(* CoDeSys 2.3.9.47 project: 3floor_2016_06_22_beta.prx *)
(* Libraries: TcEIB.lbx 16.5.14 14:12:22, TcSystemBX.lbx 11.6.12 13:56:16, TcBaseBX.lbx 10.5.06 08:50:20, standard.lbx 5.12.03 08:02:30 *)

(* Task configuration *)
TASK Standard (PRIORITY := 0, INTERVAL := T#20ms);
	MAIN
END_TASK

(* Global variable list: M_Var_1 *)
VAR_GLOBAL

	komora_l_adr: 				EIB_GROUP_ADDR:= (MAIN:=1, SUB_MAIN:=1, NUMBER:=10);
	su1_l_adr: 					EIB_GROUP_ADDR:= (MAIN:=1, SUB_MAIN:=1, NUMBER:=11);
	topochna_l_adr:	 			EIB_GROUP_ADDR:= (MAIN:=1, SUB_MAIN:=1, NUMBER:=12);
	su2_bra_adr:	 			EIB_GROUP_ADDR:= (MAIN:=1, SUB_MAIN:=1, NUMBER:=13);
	su2_l_adr:	 				EIB_GROUP_ADDR:= (MAIN:=1, SUB_MAIN:=1, NUMBER:=14);
	su1_rakovyna_adr:	 		EIB_GROUP_ADDR:= (MAIN:=1, SUB_MAIN:=1, NUMBER:=15);
	su2_dush_adr:	 			EIB_GROUP_ADDR:= (MAIN:=1, SUB_MAIN:=1, NUMBER:=16);
	dush_adr:	 				EIB_GROUP_ADDR:= (MAIN:=1, SUB_MAIN:=1, NUMBER:=17);
	kuhnya1_adr:	 			EIB_GROUP_ADDR:= (MAIN:=1, SUB_MAIN:=1, NUMBER:=18);
	vitalnya_smugy1_adr: 		EIB_GROUP_ADDR:= (MAIN:=1, SUB_MAIN:=1, NUMBER:=19);
	vitalnya_l_adr: 				EIB_GROUP_ADDR:= (MAIN:=1, SUB_MAIN:=1, NUMBER:=20);
	vitalnya_prokladka_adr: 		EIB_GROUP_ADDR:= (MAIN:=1, SUB_MAIN:=1, NUMBER:=21);
	terassa_stina_adr: 			EIB_GROUP_ADDR:= (MAIN:=1, SUB_MAIN:=1, NUMBER:=22);
	pidval_shody_adr: 			EIB_GROUP_ADDR:= (MAIN:=1, SUB_MAIN:=1, NUMBER:=23);
	skhody2pov_adr: 			EIB_GROUP_ADDR:= (MAIN:=1, SUB_MAIN:=1, NUMBER:=24);
	tambur_l_adr:				EIB_GROUP_ADDR:= (MAIN:=1, SUB_MAIN:=1, NUMBER:=25);
	vent_su1_adr: 				EIB_GROUP_ADDR:= (MAIN:=1, SUB_MAIN:=1, NUMBER:=26);
	vent_kuh_low_adr: 			EIB_GROUP_ADDR:= (MAIN:=1, SUB_MAIN:=1, NUMBER:=27);
	vent_dush_adr: 				EIB_GROUP_ADDR:= (MAIN:=1, SUB_MAIN:=1, NUMBER:=28);
	vent_komora_adr: 			EIB_GROUP_ADDR:= (MAIN:=1, SUB_MAIN:=1, NUMBER:=29);
	vent_kuh_high_adr: 			EIB_GROUP_ADDR:= (MAIN:=1, SUB_MAIN:=1, NUMBER:=30);


	komora_l_status_adr: 				EIB_GROUP_ADDR:= (MAIN:=1, SUB_MAIN:=1, NUMBER:=110);
	su1_l_status_adr: 					EIB_GROUP_ADDR:= (MAIN:=1, SUB_MAIN:=1, NUMBER:=111);
	topochna_l_status_adr:	 			EIB_GROUP_ADDR:= (MAIN:=1, SUB_MAIN:=1, NUMBER:=112);
	su2_bra_status_adr:	 				EIB_GROUP_ADDR:= (MAIN:=1, SUB_MAIN:=1, NUMBER:=113);
	su2_l_status_adr:	 				EIB_GROUP_ADDR:= (MAIN:=1, SUB_MAIN:=1, NUMBER:=114);
	su1_rakovyna_status_adr:	 		EIB_GROUP_ADDR:= (MAIN:=1, SUB_MAIN:=1, NUMBER:=115);
	su2_dush_status_adr:	 			EIB_GROUP_ADDR:= (MAIN:=1, SUB_MAIN:=1, NUMBER:=116);
	dush_status_adr:	 				EIB_GROUP_ADDR:= (MAIN:=1, SUB_MAIN:=1, NUMBER:=117);
	kuhnya1_status_adr:	 				EIB_GROUP_ADDR:= (MAIN:=1, SUB_MAIN:=1, NUMBER:=118);
	vitalnya_smugy1_status_adr: 			EIB_GROUP_ADDR:= (MAIN:=1, SUB_MAIN:=1, NUMBER:=119);
	vitalnya_l_status_adr: 				EIB_GROUP_ADDR:= (MAIN:=1, SUB_MAIN:=1, NUMBER:=120);
	vitalnya_prokladka_status_adr: 		EIB_GROUP_ADDR:= (MAIN:=1, SUB_MAIN:=1, NUMBER:=121);
	terassa_stina_status_adr: 			EIB_GROUP_ADDR:= (MAIN:=1, SUB_MAIN:=1, NUMBER:=122);
	pidval_shody_status_adr: 			EIB_GROUP_ADDR:= (MAIN:=1, SUB_MAIN:=1, NUMBER:=123);
	skhody2pov_status_adr: 				EIB_GROUP_ADDR:= (MAIN:=1, SUB_MAIN:=1, NUMBER:=124);
	tambur_l_status_adr:					EIB_GROUP_ADDR:= (MAIN:=1, SUB_MAIN:=1, NUMBER:=125);
	vent_su1_status_adr: 				EIB_GROUP_ADDR:= (MAIN:=1, SUB_MAIN:=1, NUMBER:=126);
	vent_kuh_low_status_adr: 			EIB_GROUP_ADDR:= (MAIN:=1, SUB_MAIN:=1, NUMBER:=127);
	vent_dush_status_adr: 				EIB_GROUP_ADDR:= (MAIN:=1, SUB_MAIN:=1, NUMBER:=128);
	vent_komora_status_adr: 			EIB_GROUP_ADDR:= (MAIN:=1, SUB_MAIN:=1, NUMBER:=129);
	vent_kuh_high_status_adr: 			EIB_GROUP_ADDR:= (MAIN:=1, SUB_MAIN:=1, NUMBER:=130);



	fb_komora_l_send_status_ex: 			EIB_BIT_SEND_EX;
	fb_su1_l_send_status_ex: 				EIB_BIT_SEND_EX;
	fb_topochna_l_send_status_ex: 			EIB_BIT_SEND_EX;
	fb_su2_bra_send_status_ex: 				EIB_BIT_SEND_EX;
	fb_topochna2_l_send_status_ex: 		EIB_BIT_SEND_EX;
	fb_su2_l_send_status_ex: 				EIB_BIT_SEND_EX;
	fb_su1_rakovyna_send_status_ex: 		EIB_BIT_SEND_EX;
	fb_su2_dush_send_status_ex: 			EIB_BIT_SEND_EX;
	fb_dush_send_status_ex: 				EIB_BIT_SEND_EX;
	fb_vitalnya_smugy2_send_status_ex: 		EIB_BIT_SEND_EX;
	fb_su2_polytsi_send_status_ex: 			EIB_BIT_SEND_EX;
	fb_kuhnya1_send_status_ex: 			EIB_BIT_SEND_EX;
	fb_kuhnya2_send_status_ex: 			EIB_BIT_SEND_EX;
	fb_vitalnya_smugy1_send_status_ex: 		EIB_BIT_SEND_EX;
	fb_vitalnya_l_send_status_ex: 			EIB_BIT_SEND_EX;
	fb_vitalnya_prokladka_send_status_ex: 	EIB_BIT_SEND_EX;
	fb_terassa_stina_send_status_ex: 		EIB_BIT_SEND_EX;
	fb_pidval_shody_send_status_ex: 		EIB_BIT_SEND_EX;
	fb_skhody2pov_send_status_ex: 			EIB_BIT_SEND_EX;
	fb_tambur_l_send_status_ex: 			EIB_BIT_SEND_EX;
	fb_vent_su1_send_status_ex: 			EIB_BIT_SEND_EX;
	fb_vent_kuh_low_send_status_ex: 		EIB_BIT_SEND_EX;
	fb_vent_dush_send_status_ex: 			EIB_BIT_SEND_EX;
	fb_vent_komora_send_status_ex: 		EIB_BIT_SEND_EX;
	fb_vent_kuh_high_send_status_ex: 		EIB_BIT_SEND_EX;

	fb_komora_l_read: 			EIB_BIT_REC;
	fb_su1_l_read: 				EIB_BIT_REC;
	fb_topochna_l_read: 		EIB_BIT_REC;
	fb_su2_bra_read: 			EIB_BIT_REC;
	fb_topochna2_l_read: 		EIB_BIT_REC;
	fb_su2_l_read: 				EIB_BIT_REC;
	fb_su1_rakovyna_read: 		EIB_BIT_REC;
	fb_su2_dush_read: 			EIB_BIT_REC;
	fb_dush_read: 				EIB_BIT_REC;
	fb_vitalnya_smugy2_read: 	EIB_BIT_REC;
	fb_su2_polytsi_read: 		EIB_BIT_REC;
	fb_kuhnya1_read: 			EIB_BIT_REC;
	fb_kuhnya2_read: 			EIB_BIT_REC;
	fb_vitalnya_smugy1_read: 	EIB_BIT_REC;
	fb_vitalnya_l_read: 			EIB_BIT_REC;
	fb_vitalnya_prokladka_read: 	EIB_BIT_REC;
	fb_terassa_stina_read: 		EIB_BIT_REC;
	fb_pidval_shody_read: 		EIB_BIT_REC;
	fb_skhody2pov_read: 		EIB_BIT_REC;
	fb_tambur_l_read: 			EIB_BIT_REC;
	fb_vent_su1_read: 			EIB_BIT_REC;
	fb_vent_kuh_low_read: 		EIB_BIT_REC;
	fb_vent_dush_read: 			EIB_BIT_REC;
	fb_vent_komora_read: 		EIB_BIT_REC;
	fb_vent_kuh_high_read: 		EIB_BIT_REC;

	moove_garderob				AT%MX100.0:BOOL;
	moove_tambur					AT%MX100.1:BOOL;
	moove_dytjacha					AT%MX100.2:BOOL;
	moove_spalnya					AT%MX100.3:BOOL;
	moove_korydor					AT%MX100.4:BOOL;
	moove_skhody					AT%MX100.5:BOOL;

	komora_l 						AT%MX100.0:BOOL;
	su1_l 							AT%MX100.1:BOOL;
	topochna_l 						AT%MX100.2:BOOL;
	su2_bra	 						AT%MX100.3:BOOL;
	su2_l 							AT%MX100.4:BOOL;
	su1_rakovyna 					AT%MX100.5:BOOL;
	su2_dush 						AT%MX100.6:BOOL;
	dush 							AT%MX100.7:BOOL;

	kuhnya1	 					AT%MX101.0:BOOL;
	vitalnya_smugy1 				AT%MX101.1:BOOL;
	vitalnya_l 						AT%MX101.2:BOOL;
	vitalnya_prokladka 				AT%MX101.3:BOOL;
	terassa_stina	 				AT%MX101.4:BOOL;
	pidval_shody	 				AT%MX101.5:BOOL;
	skhody2pov 					AT%MX101.6:BOOL;
	tambur_l 						AT%MX101.7:BOOL;

	vent_su1 						AT%MX102.0:BOOL;
	vent_kuh_low 					AT%MX102.1:BOOL;
	vent_dush 						AT%MX102.2:BOOL;
	vent_komora 					AT%MX102.3:BOOL;
	vent_kuh_high 					AT%MX102.4:BOOL;

END_VAR

(* Global variable list: M_Var_2 *)
VAR_GLOBAL
	balkon_peryla_adr: EIB_GROUP_ADDR:=(MAIN:=1, SUB_MAIN:=4, NUMBER:=9);
	kino_l_adr: EIB_GROUP_ADDR:= (MAIN:=1, SUB_MAIN:=4, NUMBER:=10);
	balkon_bra_adr:	 EIB_GROUP_ADDR:= (MAIN:=1, SUB_MAIN:=4, NUMBER:=11);
	kabinet_balkon_l_adr:	 EIB_GROUP_ADDR:= (MAIN:=1, SUB_MAIN:=4, NUMBER:=12);
	balkon_adr:	 EIB_GROUP_ADDR:= (MAIN:=1, SUB_MAIN:=4, NUMBER:=13);
	korydor1_adr:	 EIB_GROUP_ADDR:= (MAIN:=1, SUB_MAIN:=4, NUMBER:=14);
	kino_bra_adr:	 EIB_GROUP_ADDR:= (MAIN:=1, SUB_MAIN:=4, NUMBER:=15);
	korydor2_adr:	 EIB_GROUP_ADDR:= (MAIN:=1, SUB_MAIN:=4, NUMBER:=16);
	studio_pidsvitka_adr:	 EIB_GROUP_ADDR:= (MAIN:=1, SUB_MAIN:=4, NUMBER:=17);
	skhody2_3_adr:	 EIB_GROUP_ADDR:= (MAIN:=1, SUB_MAIN:=4, NUMBER:=18);
	studio_l_adr:	 EIB_GROUP_ADDR:= (MAIN:=1, SUB_MAIN:=4, NUMBER:=19);
	kabinet_pidsvitka_kolo_adr:	 EIB_GROUP_ADDR:= (MAIN:=1, SUB_MAIN:=4, NUMBER:=20);
	kabinet_svitlo_adr:	 EIB_GROUP_ADDR:= (MAIN:=1, SUB_MAIN:=4, NUMBER:=21);
	stend_adr:	 EIB_GROUP_ADDR:= (MAIN:=1, SUB_MAIN:=4, NUMBER:=22);
	kabinet_kobra_adr:	 EIB_GROUP_ADDR:= (MAIN:=1, SUB_MAIN:=4, NUMBER:=23);
	skhody_peryla_adr:	 EIB_GROUP_ADDR:= (MAIN:=1, SUB_MAIN:=4, NUMBER:=24);
	tambur2_adr:	 EIB_GROUP_ADDR:= (MAIN:=1, SUB_MAIN:=4, NUMBER:=25);

	fb_balkon_peryla_send: EIB_BIT_SEND_MANUAL;
	fb_kino_l_send:  EIB_BIT_SEND_manual;
	fb_balkon_bra_send: EIB_BIT_SEND_manual;
	fb_kabinet_balkon_l_send:  EIB_BIT_SEND_manual;
	fb_balkon_send:	EIB_BIT_SEND_manual;
	fb_korydor1_send:	 EIB_BIT_SEND_manual;
	fb_kino_bra_send:	EIB_BIT_SEND_manual;
	fb_korydor2_send:	EIB_BIT_SEND_manual;
	fb_studio_pidsvitka_send: EIB_BIT_SEND_MANUAL;
	fb_skhody2_3_send:	  EIB_BIT_SEND_MANUAL;
	fb_studio_l_send:	 EIB_BIT_SEND_manual;
	fb_kabinet_pidsvitka_kolo_send:	EIB_BIT_SEND_MANUAL;
	fb_kabinet_svitlo_send:	EIB_BIT_SEND_manual;
	fb_stend_send:  EIB_BIT_SEND_manual;
	fb_kabinet_kobra_send:  EIB_BIT_SEND_manual;
	fb_skhody_peryla_send:  EIB_BIT_SEND_MANUAL;
	fb_tambur2_send: EIB_BIT_SEND_MANUAL;
	fb_balkon_peryla_read: EIB_BIT_REC;
	fb_kino_l_read:  EIB_BIT_rec;
	fb_balkon_bra_read: EIB_BIT_rec;
	fb_kabinet_balkon_l_read:  EIB_BIT_rec;
	fb_balkon_read:	EIB_BIT_rec;
	fb_korydor1_read:	 EIB_BIT_rec;
	fb_kino_bra_read:	EIB_BIT_rec;
	fb_korydor2_read:	EIB_BIT_rec;
	fb_studio_pidsvitka_read: EIB_BIT_rec;
	fb_skhody2_3_read:	  EIB_BIT_REC;
	fb_studio_l_read:	 EIB_BIT_rec;
	fb_kabinet_pidsvitka_kolo_read:	EIB_BIT_REC;
	fb_kabinet_svitlo_read:	EIB_BIT_REC;
	fb_stend_read:  EIB_BIT_rec;
	fb_kabinet_kobra_read:  EIB_BIT_rec;
	fb_skhody_peryla_read:  EIB_BIT_REC;
	fb_tambur2_read: EIB_BIT_REC;


	eib_shtory_kino, eib_tul_kino: EIB_BIT_REC; (*ловлять в мережі смартбаса телеграмки для штор і тюлей*)
	eib_shtory_kabinet, eib_tul_kabinet: EIB_BIT_REC;

	fb_eib_shtory_kino_move:EIB_BIT_REC;
	fb_eib_shtory_kino_position:EIB_8BIT_SIGN_REC;
	fb_eib_shtory_kino_actualPosition:EIB_8BIT_SIGN_SEND;

	fb_eib_tul_kino_move:EIB_BIT_REC;
	fb_eib_tul_kino_position:EIB_8BIT_SIGN_REC;
	fb_eib_tul_kino_actualPosition:EIB_8BIT_SIGN_SEND;

	fb_eib_shtory_kabinet_move:EIB_BIT_REC;
	fb_eib_shtory_kabinet_position:EIB_8BIT_SIGN_REC;
	fb_eib_shtory_kabinet_actualPosition:EIB_8BIT_SIGN_SEND;

	fb_eib_tul_kabinet_move:EIB_BIT_REC;
	fb_eib_tul_kabinet_position:EIB_8BIT_SIGN_REC;
	fb_eib_tul_kabinet_actualPosition:EIB_8BIT_SIGN_SEND;



	balkon_peryla					AT%MX200.0:BOOL;
	kino_l							AT%MX200.1:BOOL;
	balkon_bra						AT%MX200.2:BOOL;
	kabinet_balkon_l					AT%MX200.3:BOOL;
	balkon							AT%MX200.4:BOOL;
	korydor1							AT%MX200.5:BOOL;
	kino_bra							AT%MX200.6:BOOL;
	korydor2							AT%MX200.7:BOOL;
	studio_pidsvitka					AT%MX201.0:BOOL;
	skhody2_3						AT%MX201.1:BOOL;
	studio_l							AT%MX201.2:BOOL;
	kabinet_pidsvitka_kolo				AT%MX201.3:BOOL;
	kabinet_svitlo						AT%MX201.4:BOOL;
	kabinet_kobra					AT%MX201.5:BOOL;
	tambur2							AT%MX201.6:BOOL;
	stend							AT%MX201.7:BOOL;
	skhody_peryla					AT%MX202.0:BOOL;

	kino_shtory_status					AT%MX202.1:BOOL;
	kino_tul_status					AT%MX202.2:BOOL;
	kabinet_shtory_status				AT%MX202.3:BOOL;
	kabinet_tul_status					AT%MX202.4:BOOL;

	collector_kabinet1					AT%MX203.0:BOOL;
	collector_kabinet2					AT%MX203.1:BOOL;
	collector_studio1					AT%MX203.2:BOOL;
	collector_studio2					AT%MX203.3:BOOL;

	fancoil_kabinet_low				AT%MX203.4:BOOL;
	fancoil_kabinet_med				AT%MX203.5:BOOL;
	fancoil_kabinet_high				AT%MX203.6:BOOL;

	fancoil_kino_low					AT%MX203.7:BOOL;
	fancoil_kino_med					AT%MX204.0:BOOL;
	fancoil_kino_high					AT%MX204.1:BOOL;


	kino_shtory_ActualPosition		AT%MB205:USINT;
	kino_tul_ActualPosition			AT%MB206:USINT;
	kabinet_shtory_ActualPosition	AT%MB207:USINT;
	kabinet_tul_ActualPosition		AT%MB208:USINT;
END_VAR

(* Global variable list: M_Var_4 *)
VAR_GLOBAL

	derevo_vidpochynok1_adr:	 	EIB_GROUP_ADDR:= (MAIN:=1, SUB_MAIN:=7, NUMBER:=22);
	derevo_vidpochynok2_adr:	 	EIB_GROUP_ADDR:= (MAIN:=1, SUB_MAIN:=7, NUMBER:=1);
	derevo_veranda_adr:	 		EIB_GROUP_ADDR:= (MAIN:=1, SUB_MAIN:=7, NUMBER:=2);
	derevo_veranda_zovn_adr:	 	EIB_GROUP_ADDR:= (MAIN:=1, SUB_MAIN:=7, NUMBER:=3);
	derevo_vhid_zovn_adr:	 		EIB_GROUP_ADDR:= (MAIN:=1, SUB_MAIN:=7, NUMBER:=4);
	derevo_sauna_adr:	 			EIB_GROUP_ADDR:= (MAIN:=1, SUB_MAIN:=7, NUMBER:=5);
	derevo_vhid_adr:				EIB_GROUP_ADDR:= (MAIN:=1, SUB_MAIN:=7, NUMBER:=6);
	derevo_kotel_adr:		 		EIB_GROUP_ADDR:= (MAIN:=1, SUB_MAIN:=7, NUMBER:=7);
	derevo_korydor_adr:		 		EIB_GROUP_ADDR:= (MAIN:=1, SUB_MAIN:=7, NUMBER:=8);
	derevo_sinna_adr:		 		EIB_GROUP_ADDR:= (MAIN:=1, SUB_MAIN:=7, NUMBER:=9);
	derevo_hamam_adr:		 		EIB_GROUP_ADDR:= (MAIN:=1, SUB_MAIN:=7, NUMBER:=10);
	derevo_kuhnya_adr:	 			EIB_GROUP_ADDR:= (MAIN:=1, SUB_MAIN:=7, NUMBER:=11);
	derevo_bassein1_adr:			EIB_GROUP_ADDR:= (MAIN:=1, SUB_MAIN:=7, NUMBER:=12);
	derevo_bassein_lampa_adr:		EIB_GROUP_ADDR:= (MAIN:=1, SUB_MAIN:=7, NUMBER:=13);
	derevo_spalnya2_adr:			EIB_GROUP_ADDR:= (MAIN:=1, SUB_MAIN:=7, NUMBER:=14);
	derevo_terassa_adr:				EIB_GROUP_ADDR:= (MAIN:=1, SUB_MAIN:=7, NUMBER:=15);
	derevo_dush_adr:	 			EIB_GROUP_ADDR:= (MAIN:=1, SUB_MAIN:=7, NUMBER:=16);
	derevo_wc_adr:					EIB_GROUP_ADDR:= (MAIN:=1, SUB_MAIN:=7, NUMBER:=17);
	derevo_spalnya_verh_adr:		EIB_GROUP_ADDR:= (MAIN:=1, SUB_MAIN:=7, NUMBER:=18);
	derevo_spalnya1_adr:			EIB_GROUP_ADDR:= (MAIN:=1, SUB_MAIN:=7, NUMBER:=19);
	derevo_spalnya_su_adr:			EIB_GROUP_ADDR:= (MAIN:=1, SUB_MAIN:=7, NUMBER:=20);
	derevo_garderob_adr:			EIB_GROUP_ADDR:= (MAIN:=1, SUB_MAIN:=7, NUMBER:=21);
	derevo_dush2_adr:				EIB_GROUP_ADDR:= (MAIN:=1, SUB_MAIN:=7, NUMBER:=23);

	derevo_vidpochynok1_status_adr:	 	EIB_GROUP_ADDR:= (MAIN:=1, SUB_MAIN:=7, NUMBER:=122);
	derevo_vidpochynok2_status_adr:	 	EIB_GROUP_ADDR:= (MAIN:=1, SUB_MAIN:=7, NUMBER:=101);
	derevo_veranda_status_adr:	 			EIB_GROUP_ADDR:= (MAIN:=1, SUB_MAIN:=7, NUMBER:=102);
	derevo_veranda_zovn_status_adr:	 	EIB_GROUP_ADDR:= (MAIN:=1, SUB_MAIN:=7, NUMBER:=103);
	derevo_vhid_zovn_status_adr:	 		EIB_GROUP_ADDR:= (MAIN:=1, SUB_MAIN:=7, NUMBER:=104);
	derevo_sauna_status_adr:	 			EIB_GROUP_ADDR:= (MAIN:=1, SUB_MAIN:=7, NUMBER:=105);
	derevo_vhid_status_adr:					EIB_GROUP_ADDR:= (MAIN:=1, SUB_MAIN:=7, NUMBER:=106);
	derevo_kotel_status_adr:		 		EIB_GROUP_ADDR:= (MAIN:=1, SUB_MAIN:=7, NUMBER:=107);
	derevo_korydor_status_adr:		 		EIB_GROUP_ADDR:= (MAIN:=1, SUB_MAIN:=7, NUMBER:=108);
	derevo_sinna_status_adr:		 		EIB_GROUP_ADDR:= (MAIN:=1, SUB_MAIN:=7, NUMBER:=109);
	derevo_hamam_status_adr:		 		EIB_GROUP_ADDR:= (MAIN:=1, SUB_MAIN:=7, NUMBER:=110);
	derevo_kuhnya_status_adr:	 			EIB_GROUP_ADDR:= (MAIN:=1, SUB_MAIN:=7, NUMBER:=111);
	derevo_bassein1_status_adr:				EIB_GROUP_ADDR:= (MAIN:=1, SUB_MAIN:=7, NUMBER:=112);
	derevo_bassein_lampa_status_adr:		EIB_GROUP_ADDR:= (MAIN:=1, SUB_MAIN:=7, NUMBER:=113);
	derevo_spalnya2_status_adr:				EIB_GROUP_ADDR:= (MAIN:=1, SUB_MAIN:=7, NUMBER:=114);
	derevo_terassa_status_adr:				EIB_GROUP_ADDR:= (MAIN:=1, SUB_MAIN:=7, NUMBER:=115);
	derevo_dush_status_adr:	 			EIB_GROUP_ADDR:= (MAIN:=1, SUB_MAIN:=7, NUMBER:=116);
	derevo_wc_status_adr:					EIB_GROUP_ADDR:= (MAIN:=1, SUB_MAIN:=7, NUMBER:=117);
	derevo_spalnya_verh_status_adr:		EIB_GROUP_ADDR:= (MAIN:=1, SUB_MAIN:=7, NUMBER:=118);
	derevo_spalnya1_status_adr:				EIB_GROUP_ADDR:= (MAIN:=1, SUB_MAIN:=7, NUMBER:=119);
	derevo_spalnya_su_status_adr:			EIB_GROUP_ADDR:= (MAIN:=1, SUB_MAIN:=7, NUMBER:=120);
	derevo_garderob_status_adr:				EIB_GROUP_ADDR:= (MAIN:=1, SUB_MAIN:=7, NUMBER:=121);
	derevo_dush2_status_adr:				EIB_GROUP_ADDR:= (MAIN:=1, SUB_MAIN:=7, NUMBER:=123);

	fb_derevo_vidpochynok1_send_status_ex: 		EIB_BIT_SEND_EX;
	fb_derevo_vidpochynok2_send_status_ex: 		EIB_BIT_SEND_EX;
	fb_derevo_veranda_send_status_ex: 				EIB_BIT_SEND_EX;
	fb_derevo_veranda_zovn_send_status_ex: 		EIB_BIT_SEND_EX;
	fb_derevo_vhid_zovn_send_status_ex: 			EIB_BIT_SEND_EX;
	fb_derevo_sauna_send_status_ex: 				EIB_BIT_SEND_EX;
	fb_derevo_vhid_send_status_ex: 				EIB_BIT_SEND_EX;
	fb_derevo_kotel_send_status_ex: 				EIB_BIT_SEND_EX;
	fb_derevo_korydor_send_status_ex: 				EIB_BIT_SEND_EX;
	fb_derevo_sinna_send_status_ex: 				EIB_BIT_SEND_EX;
	fb_derevo_hamam_send_status_ex: 				EIB_BIT_SEND_EX;
	fb_derevo_kuhnya_send_status_ex: 				EIB_BIT_SEND_EX;
	fb_derevo_bassein1_send_status_ex: 			EIB_BIT_SEND_EX;
	fb_derevo_bassein_lampa_send_status_ex: 		EIB_BIT_SEND_EX;
	fb_derevo_spalnya2_send_status_ex: 			EIB_BIT_SEND_EX;
	fb_derevo_terassa_send_status_ex: 				EIB_BIT_SEND_EX;
	fb_derevo_dush_send_status_ex: 				EIB_BIT_SEND_EX;
	fb_derevo_wc_send_status_ex: 					EIB_BIT_SEND_EX;
	fb_derevo_spalnya_verh_send_status_ex: 		EIB_BIT_SEND_EX;
	fb_derevo_spalnya1_send_status_ex: 			EIB_BIT_SEND_EX;
	fb_derevo_spalnya_su_send_status_ex: 			EIB_BIT_SEND_EX;
	fb_derevo_garderob_send_status_ex: 			EIB_BIT_SEND_EX;
	fb_derevo_dush2_send_status_ex: 				EIB_BIT_SEND_EX;

	fb_derevo_vidpochynok1_read: 		EIB_BIT_REC;
	fb_derevo_vidpochynok2_read: 		EIB_BIT_REC;
	fb_derevo_veranda_read: 			EIB_BIT_REC;
	fb_derevo_veranda_zovn_read: 		EIB_BIT_REC;
	fb_derevo_vhid_zovn_read: 			EIB_BIT_REC;
	fb_derevo_sauna_read: 				EIB_BIT_REC;
	fb_derevo_vhid_read: 				EIB_BIT_REC;
	fb_derevo_kotel_read: 				EIB_BIT_REC;
	fb_derevo_korydor_read:				EIB_BIT_REC;
	fb_derevo_sinna_read: 				EIB_BIT_REC;
	fb_derevo_hamam_read: 			EIB_BIT_REC;
	fb_derevo_kuhnya_read: 			EIB_BIT_REC;
	fb_derevo_bassein1_read: 			EIB_BIT_REC;
	fb_derevo_bassein_lampa_read: 		EIB_BIT_REC;
	fb_derevo_spalnya2_read: 			EIB_BIT_REC;
	fb_derevo_terassa_read: 			EIB_BIT_REC;
	fb_derevo_dush_read: 				EIB_BIT_REC;
	fb_derevo_wc_read: 				EIB_BIT_REC;
	fb_derevo_spalnya_verh_read: 		EIB_BIT_REC;
	fb_derevo_spalnya1_read: 			EIB_BIT_REC;
	fb_derevo_spalnya_su_read: 		EIB_BIT_REC;
	fb_derevo_garderob_read: 			EIB_BIT_REC;
	fb_derevo_dush2_read: 				EIB_BIT_REC;

	derevo_vidpochynok1 		AT %MX400.0:	 BOOL;
	derevo_vidpochynok2 		AT %MX400.1:	 BOOL;
	derevo_veranda 			AT %MX400.2:	 BOOL;
	derevo_veranda_zovn 		AT %MX400.3:	 BOOL;
	derevo_vhid_zovn 			AT %MX400.4:	 BOOL;
	derevo_sauna 				AT %MX400.5:	 BOOL;
	derevo_vhid					AT %MX400.6:	 BOOL;
	derevo_kotel 				AT %MX400.7:	 BOOL;
	derevo_korydor 				AT %MX401.0:	 BOOL;
	derevo_sinna 				AT %MX401.1:	 BOOL;
	derevo_hamam 				AT %MX401.2:	 BOOL;
	derevo_kuhnya 				AT %MX401.3:	 BOOL;
	derevo_bassein1			AT %MX401.4:	 BOOL;
	derevo_bassein_lampa		AT %MX401.5:	 BOOL;
	derevo_spalnya2			AT %MX401.6:	 BOOL;
	derevo_terassa 				AT %MX401.7:	 BOOL;
	derevo_dush 				AT %MX402.0:	 BOOL;
	derevo_wc 					AT %MX402.1:	 BOOL;
	derevo_spalnya_verh		AT %MX402.2:	 BOOL;
	derevo_spalnya1 			AT %MX402.3:	 BOOL;
	derevo_spalnya_su 			AT %MX402.4:	 BOOL;
	derevo_garderob 			AT %MX402.5:	 BOOL;
	derevo_dush2				AT %MX402.6:	 BOOL;
END_VAR

(* Global variable list: main *)
VAR_GLOBAL


	bDarkOutside: BOOL;
	fb_KL6301_0: KL6301; (* EIB functonblock *)
	system_time:timestruct;

	VITALNYA_HVAC: ROOM_HVAC;
	SPALNYA_HVAC: ROOM_HVAC;
	DYTJACHA_HVAC: ROOM_HVAC;
	KINO_HVAC:ROOM_HVAC;
	STUDIO_HVAC: ROOM_HVAC;
	KABINET_HVAC:ROOM_HVAC;

	heating_mode:BOOL:=TRUE; (*false means COOLING*)

(*global parameters eib adresses*)
	heating_mode_addr:EIB_GROUP_ADDR:= (MAIN:=1, SUB_MAIN:=2, NUMBER:=10);

(*adresses for Temperatures from HDL panels *)
	vitalnya_T_EIB_addr: EIB_GROUP_ADDR:= (MAIN:=1, SUB_MAIN:=1, NUMBER:=0);
	kino_T_EIB_addr: EIB_GROUP_ADDR:= (MAIN:=1, SUB_MAIN:=2, NUMBER:=0);
	studio_T_EIB_addr: EIB_GROUP_ADDR:= (MAIN:=1, SUB_MAIN:=3, NUMBER:=0);
	kabinet_T_EIB_addr: EIB_GROUP_ADDR:= (MAIN:=1, SUB_MAIN:=4, NUMBER:=0);
	dytjacha_T_EIB_addr: EIB_GROUP_ADDR:= (MAIN:=1, SUB_MAIN:=5, NUMBER:=0);
	spalnya_T_EIB_addr: EIB_GROUP_ADDR:= (MAIN:=1, SUB_MAIN:=6, NUMBER:=0);
	out_t_EIB_addr:eib_group_addr:=(main:=1,sub_main:=7,number:=0);
(*adresses for actual setpoint from eib_port *)
	vitalnya_actual_setpoint_addr: EIB_GROUP_ADDR:= (MAIN:=1, SUB_MAIN:=1, NUMBER:=5);
	kino_actual_setpoint_addr: EIB_GROUP_ADDR:= (MAIN:=1, SUB_MAIN:=2, NUMBER:=5);
	studio_actual_setpoint_addr: EIB_GROUP_ADDR:= (MAIN:=1, SUB_MAIN:=3, NUMBER:=5);
	kabinet_actual_setpoint_addr: EIB_GROUP_ADDR:= (MAIN:=1, SUB_MAIN:=4, NUMBER:=5);
	dytjacha_actual_setpoint_addr: EIB_GROUP_ADDR:= (MAIN:=1, SUB_MAIN:=5, NUMBER:=5);
	spalnya_actual_setpoint_addr: EIB_GROUP_ADDR:= (MAIN:=1, SUB_MAIN:=6, NUMBER:=5);
(*adresses for current speed and setpoint of cooling mode from HDL panels *)
	vitalnya_cooling_EIB_addr: EIB_GROUP_ADDR:= (MAIN:=1, SUB_MAIN:=1, NUMBER:=1);
	kino_cooling_EIB_addr: EIB_GROUP_ADDR:= (MAIN:=1, SUB_MAIN:=2, NUMBER:=1);
	studio_cooling_EIB_addr: EIB_GROUP_ADDR:= (MAIN:=1, SUB_MAIN:=3, NUMBER:=1);
	kabinet_cooling_EIB_addr: EIB_GROUP_ADDR:= (MAIN:=1, SUB_MAIN:=4, NUMBER:=1);
	dytjacha_cooling_EIB_addr: EIB_GROUP_ADDR:= (MAIN:=1, SUB_MAIN:=5, NUMBER:=1);
	spalnya_cooling_EIB_addr: EIB_GROUP_ADDR:= (MAIN:=1, SUB_MAIN:=6, NUMBER:=1);
(*adresses for current speed and setpoint of heating mode from HDL panels *)
	vitalnya_heating_EIB_addr: EIB_GROUP_ADDR:= (MAIN:=1, SUB_MAIN:=1, NUMBER:=2);
	kino_heating_EIB_addr: EIB_GROUP_ADDR:= (MAIN:=1, SUB_MAIN:=2, NUMBER:=2);
	studio_heating_EIB_addr: EIB_GROUP_ADDR:= (MAIN:=1, SUB_MAIN:=3, NUMBER:=2);
	kabinet_heating_EIB_addr: EIB_GROUP_ADDR:= (MAIN:=1, SUB_MAIN:=4, NUMBER:=2);
	dytjacha_heating_EIB_addr: EIB_GROUP_ADDR:= (MAIN:=1, SUB_MAIN:=5, NUMBER:=2);
	spalnya_heating_EIB_addr: EIB_GROUP_ADDR:= (MAIN:=1, SUB_MAIN:=6, NUMBER:=2);

(*adresses for current speed of fan mode from HDL panels *)
	vitalnya_fan_EIB_addr: EIB_GROUP_ADDR:= (MAIN:=1, SUB_MAIN:=1, NUMBER:=3);
	kino_fan_EIB_addr: EIB_GROUP_ADDR:= (MAIN:=1, SUB_MAIN:=2, NUMBER:=3);
	studio_fan_EIB_addr: EIB_GROUP_ADDR:= (MAIN:=1, SUB_MAIN:=3, NUMBER:=3);
	kabinet_fan_EIB_addr: EIB_GROUP_ADDR:= (MAIN:=1, SUB_MAIN:=4, NUMBER:=3);
	dytjacha_fan_EIB_addr: EIB_GROUP_ADDR:= (MAIN:=1, SUB_MAIN:=5, NUMBER:=3);
	spalnya_fan_EIB_addr: EIB_GROUP_ADDR:= (MAIN:=1, SUB_MAIN:=6, NUMBER:=3);

(*adresses for FCU cooling and heating signals*)
	vitalnya_FCU_cooling_ctrl_sig_EIB_addr: EIB_GROUP_ADDR:= (MAIN:=1, SUB_MAIN:=1, NUMBER:=7);
	kino_FCU_cooling_ctrl_sig_EIB_addr: EIB_GROUP_ADDR:= (MAIN:=1, SUB_MAIN:=2, NUMBER:=7);

	kabinet_FCU_cooling_ctrl_sig_EIB_addr: EIB_GROUP_ADDR:= (MAIN:=1, SUB_MAIN:=4, NUMBER:=7);
	dytjacha_FCU_cooling_ctrl_sig_EIB_addr: EIB_GROUP_ADDR:= (MAIN:=1, SUB_MAIN:=5, NUMBER:=7);
	spalnya_FCU_cooling_ctrl_sig_EIB_addr: EIB_GROUP_ADDR:= (MAIN:=1, SUB_MAIN:=6, NUMBER:=7);

	vitalnya_FCU_heating_ctrl_sig_EIB_addr: EIB_GROUP_ADDR:= (MAIN:=1, SUB_MAIN:=1, NUMBER:=6);
	kino_FCU_heating_ctrl_sig_EIB_addr: EIB_GROUP_ADDR:= (MAIN:=1, SUB_MAIN:=2, NUMBER:=6);
	kabinet_FCU_heating_ctrl_sig_EIB_addr: EIB_GROUP_ADDR:= (MAIN:=1, SUB_MAIN:=4, NUMBER:=6);
	dytjacha_FCU_heating_ctrl_sig_EIB_addr: EIB_GROUP_ADDR:= (MAIN:=1, SUB_MAIN:=5, NUMBER:=6);
	spalnya_FCU_heating_ctrl_sig_EIB_addr: EIB_GROUP_ADDR:= (MAIN:=1, SUB_MAIN:=6, NUMBER:=6);
(*adresses for FCU cooling and heating signals*)
	vitalnya_FCU_fan_speed_EIB_addr: EIB_GROUP_ADDR:= (MAIN:=1, SUB_MAIN:=1, NUMBER:=8);
	kino_FCU_fan_speed_EIB_addr: EIB_GROUP_ADDR:= (MAIN:=1, SUB_MAIN:=2, NUMBER:=8);
	studio_FCU_fan_speed_EIB_addr: EIB_GROUP_ADDR:= (MAIN:=1, SUB_MAIN:=3, NUMBER:=8);
	kabinet_FCU_fan_speed_EIB_addr: EIB_GROUP_ADDR:= (MAIN:=1, SUB_MAIN:=4, NUMBER:=8);
	dytjacha_FCU_fan_speed_EIB_addr: EIB_GROUP_ADDR:= (MAIN:=1, SUB_MAIN:=5, NUMBER:=8);
	spalnya_FCU_fan_speed_EIB_addr: EIB_GROUP_ADDR:= (MAIN:=1, SUB_MAIN:=6, NUMBER:=8);
(*adresses for damper  control and indication*)
	vitalnya_damper_EIB_addr: EIB_GROUP_ADDR:= (MAIN:=1, SUB_MAIN:=2, NUMBER:=10);
	kino_damper_EIB_addr: EIB_GROUP_ADDR:= (MAIN:=1, SUB_MAIN:=2, NUMBER:=11);
	kabinet_damper_EIB_addr: EIB_GROUP_ADDR:= (MAIN:=1, SUB_MAIN:=2, NUMBER:=12);
	dytjacha_damper_EIB_addr: EIB_GROUP_ADDR:= (MAIN:=1, SUB_MAIN:=2, NUMBER:=13);
	spalnya_damper_EIB_addr: EIB_GROUP_ADDR:= (MAIN:=1, SUB_MAIN:=2, NUMBER:=14);

(**adresses for shtory*)
	move_shtory_kino_EIB_addr: EIB_GROUP_ADDR := (MAIN:=1, SUB_MAIN:=2, NUMBER:=20);
	position_shtory_kino_EIB_addr: EIB_GROUP_ADDR := (MAIN:=1, SUB_MAIN:=2, NUMBER:=21);
	actrualPosition_shtory_kino_EIB_addr: EIB_GROUP_ADDR := (MAIN:=1, SUB_MAIN:=2, NUMBER:=22);

	move_tul_kino_EIB_addr: EIB_GROUP_ADDR := (MAIN:=1, SUB_MAIN:=2, NUMBER:=23);
	position_tul_kino_EIB_addr: EIB_GROUP_ADDR := (MAIN:=1, SUB_MAIN:=2, NUMBER:=24);
	actrualPosition_tul_kino_EIB_addr: EIB_GROUP_ADDR := (MAIN:=1, SUB_MAIN:=2, NUMBER:=25);

	move_shtory_kabinet_EIB_addr: EIB_GROUP_ADDR := (MAIN:=1, SUB_MAIN:=2, NUMBER:=26);
	position_shtory_kabinet_EIB_addr: EIB_GROUP_ADDR := (MAIN:=1, SUB_MAIN:=2, NUMBER:=27);
	actrualPosition_shtory_kabinet_EIB_addr: EIB_GROUP_ADDR := (MAIN:=1, SUB_MAIN:=2, NUMBER:=28);

	move_tul_kabinet_EIB_addr: EIB_GROUP_ADDR := (MAIN:=1, SUB_MAIN:=2, NUMBER:=29);
	position_tul_kabinet_EIB_addr: EIB_GROUP_ADDR := (MAIN:=1, SUB_MAIN:=2, NUMBER:=30);
	actrualPosition_tul_kabinet_EIB_addr: EIB_GROUP_ADDR := (MAIN:=1, SUB_MAIN:=2, NUMBER:=31);

	shtory_spalnya_EIB_addr: EIB_GROUP_ADDR := (MAIN:=1, SUB_MAIN:=6, NUMBER:=31);
	tul_spalnya_EIB_addr: EIB_GROUP_ADDR := (MAIN:=1, SUB_MAIN:=6, NUMBER:=30);
	lift_spalnya_EIB_addr: EIB_GROUP_ADDR := (MAIN:=1, SUB_MAIN:=6, NUMBER:=29);
(*eib date and time adresses*)
	eib_time_EIB_addr:eib_group_addr:=(MAIN:=1, sub_main:=3, number:=10);
	eib_date_EIB_addr:eib_group_addr:=(MAIN:=1, sub_main:=3, number:=11);
	eib_twillight_EIB_addr:eib_group_addr:=(MAIN:=1, sub_main:=3, number:=12);


(*adresses for light groups*)
	spalnya_kontrazhur_adr: EIB_GROUP_ADDR:=(MAIN:=1, SUB_MAIN:=6, NUMBER:=9);
	spalnya_balkon_adr: EIB_GROUP_ADDR:=(MAIN:=1, SUB_MAIN:=6, NUMBER:=10);
	spalnya_kulbaba_adr: EIB_GROUP_ADDR:=(MAIN:=1, SUB_MAIN:=6, NUMBER:=11);
	spalnya_kontrazhur_b_adr: EIB_GROUP_ADDR:=(MAIN:=1, SUB_MAIN:=6, NUMBER:=12);
	spalnya_kontrazhur_l_adr: EIB_GROUP_ADDR:=(MAIN:=1, SUB_MAIN:=6, NUMBER:=13);

	su3_stina_adr: EIB_GROUP_ADDR:=(MAIN:=1, SUB_MAIN:=6, NUMBER:=14);
	su3_pidsvitka_adr: EIB_GROUP_ADDR:=(MAIN:=1, SUB_MAIN:=6, NUMBER:=15);
	su3_bra_adr: EIB_GROUP_ADDR:=(MAIN:=1, SUB_MAIN:=6, NUMBER:=16);
	su3_kontrazhur_adr: EIB_GROUP_ADDR:=(MAIN:=1, SUB_MAIN:=6, NUMBER:=17);
	su3_kontrazhur_k_adr: EIB_GROUP_ADDR:=(MAIN:=1, SUB_MAIN:=6, NUMBER:=19);
	su3_lampa_adr: EIB_GROUP_ADDR:=(MAIN:=1, SUB_MAIN:=6, NUMBER:=21);

	dytjacha_adr: EIB_GROUP_ADDR:=(MAIN:=1, SUB_MAIN:=6, NUMBER:=18);
	dytjacha_bra_adr: EIB_GROUP_ADDR:=(MAIN:=1, SUB_MAIN:=6, NUMBER:=20);

	garderob_adr: EIB_GROUP_ADDR:=(MAIN:=1, SUB_MAIN:=6, NUMBER:=22);
	bar_adr: EIB_GROUP_ADDR:=(MAIN:=1, SUB_MAIN:=6, NUMBER:=23);
	korydor_skeli_adr: EIB_GROUP_ADDR:=(MAIN:=1, SUB_MAIN:=6, NUMBER:=24);
	choven_adr: EIB_GROUP_ADDR:=(MAIN:=1, SUB_MAIN:=6, NUMBER:=25);
	korydor_svitlo_adr: EIB_GROUP_ADDR:=(MAIN:=1, SUB_MAIN:=6, NUMBER:=26);
	korydor_lampa_adr: EIB_GROUP_ADDR:=(MAIN:=1, SUB_MAIN:=6, NUMBER:=27);
	serverna_adr: EIB_GROUP_ADDR:=(MAIN:=1, SUB_MAIN:=6, NUMBER:=28);



	moove_sensors_adr:EIB_GROUP_ADDR:=(MAIN:=1, SUB_MAIN:=7, NUMBER:=23);


	fb_spalnya_kontrazhur_send: EIB_BIT_SEND_manual;
	fb_spalnya_balkon_send: EIB_BIT_SEND_manual;
	fb_spalnya_kulbaba_send: EIB_BIT_SEND_manual;
	fb_spalnya_kontrazhur_b_send: EIB_BIT_SEND_manual;
	fb_spalnya_kontrazhur_l_send: EIB_BIT_SEND_manual;

	fb_su3_stina_send: EIB_BIT_SEND_MANUAL;
	fb_su3_pidsvitka_send: EIB_BIT_SEND_manual;
	fb_su3_bra_send: EIB_BIT_SEND_manual;
	fb_su3_kontrazhur_send: EIB_BIT_SEND_MANUAL;
	fb_su3_kontrazhur_k_send: EIB_BIT_SEND_manual;
	fb_su3_lampa_send: EIB_BIT_SEND_manual;

	fb_dytjacha_send: EIB_BIT_SEND_MANUAL;
	fb_dytjacha_bra_send: EIB_BIT_SEND_MANUAL;

	fb_garderob_send: EIB_BIT_SEND_manual;
	fb_bar_send: EIB_BIT_SEND_MANUAL;
	fb_korydor_skeli_send: EIB_BIT_SEND_manual;
	fb_choven_send: EIB_BIT_SEND_manual;
	fb_korydor_svitlo_send: EIB_BIT_SEND_manual;
	fb_korydor_lampa_send: EIB_BIT_SEND_manual;
	fb_serverna_send: EIB_BIT_SEND_MANUAL;

	eib_shtory, eib_tul, eib_lift: EIB_BIT_REC;

	fb_spalnya_kontrazhur_read: EIB_BIT_REC;
	fb_spalnya_balkon_read: EIB_BIT_rec;
	fb_spalnya_kulbaba_read: EIB_BIT_rec;
	fb_spalnya_kontrazhur_b_read: EIB_BIT_rec;
	fb_spalnya_kontrazhur_l_read: EIB_BIT_REC;

	fb_su3_stina_read: EIB_BIT_REC;
	fb_su3_pidsvitka_read: EIB_BIT_REC;
	fb_su3_bra_read: EIB_BIT_REC;
	fb_su3_kontrazhur_read: EIB_BIT_REC;
	fb_su3_kontrazhur_k_read: EIB_BIT_REC;
	fb_su3_lampa_read: EIB_BIT_rec;

	fb_dytjacha_read: EIB_BIT_rec;
	fb_dytjacha_bra_read: EIB_BIT_REC;

	fb_garderob_read: EIB_BIT_REC;
	fb_bar_read: EIB_BIT_REC;
	fb_korydor_skeli_read: EIB_BIT_REC;
	fb_choven_read: EIB_BIT_REC;
	fb_korydor_svitlo_read: EIB_BIT_rec;
	fb_korydor_lampa_read: EIB_BIT_REC;
	fb_serverna_read: EIB_BIT_REC;
	fb_moove_sensors_read:EIB_BIT_REC;



	tLongPress: TIME; (* затримка довгого натискання *)
	tOffDelay: TIME; (* затримка для відкладеного вимкнення *)
	ads_adr1: STRING;
	ads_adr2: STRING;
	ads_adr3: STRING;
	ads_adr4: STRING;

	data1floor: ARRAY[0..200] OF SINT;
	data2floor: ARRAY[0..300] OF SINT;
	data_derevo: ARRAY[0..300] OF SINT;

	data1floor_prev: ARRAY[0..200] OF BYTE; (*попередні значення*)
	data2floor_prev: ARRAY[0..300] OF BYTE;
	data_derevo_prev: ARRAY[0..300] OF BYTE;

	moove_sensors:BOOL;



END_VAR

(* Global variable list: physical *)
VAR_GLOBAL
	din1_1	AT %IX0.0:	BOOL;
	din1_2	AT %IX0.1:	BOOL;
	din1_3	AT %IX0.2:	BOOL;
	din1_4	AT %IX0.3:	BOOL;
	din1_5	AT %IX0.4:	BOOL;
	din1_6	AT %IX0.5:	BOOL;
	din1_7	AT %IX0.6:	BOOL;
	din1_8	AT %IX0.7:	BOOL;
	din2_1	AT %IX1.0:	BOOL;
	din2_2	AT %IX1.1:	BOOL;
	din2_3	AT %IX1.2:	BOOL;
	din2_4	AT %IX1.3:	BOOL;
	din2_5	AT %IX1.4:	BOOL;
	din2_6	AT %IX1.5:	BOOL;
	din2_7	AT %IX1.6:	BOOL;
	din2_8	AT %IX1.7:	BOOL;
	sw_garderob1	AT %IX2.0:	BOOL;
	sw_dytjacha1 	AT %IX2.1:	BOOL;
	sw_garderob2	AT %IX2.2:	BOOL;
	sw_dytjacha2		AT %IX2.3:	BOOL;
	sw_tambur3_2	AT %IX2.4:	BOOL;
	sw_korydor		AT %IX2.5:	BOOL;
	sw_tambur1		AT %IX2.6:	BOOL;
	din3_8			AT %IX2.7:	BOOL;
	sw_su2			AT %IX3.0:	BOOL;
	sw_spalnya3		AT %IX3.1:	BOOL;
	sw_su1			AT %IX3.2:	BOOL;
	sw_spalnya1		AT %IX3.3:	BOOL;
	sw_spalnya_balk	AT %IX3.4:	BOOL;
	sw_spalnya2		AT %IX3.5:	BOOL;
	sw_tambur3		AT %IX3.6:	BOOL;
	sw_spalnya4		AT %IX3.7:	BOOL;
(*dout1_1*)z_vitalnya	AT %QX0.0:	BOOL;
(*dout1_2*)z_spalnya	AT %QX0.1:	BOOL;
(*dout1_3*)z_kabinet	AT %QX0.2:	BOOL;
	dout1_4	AT %QX0.3:	BOOL;
(*dout1_5*)z_kino	AT %QX0.4:	BOOL;
	dout1_6	AT %QX0.5:	BOOL;
(*dout1_7*)z_dytjacha	AT %QX0.6:	BOOL;
	dout1_8	AT %QX0.7:	BOOL;
	dout2_1	AT %QX1.0:	BOOL;
	dout2_2	AT %QX1.1:	BOOL;
	dout2_3	AT %QX1.2:	BOOL;
	dout2_4	AT %QX1.3:	BOOL;
	dout2_5	AT %QX1.4:	BOOL;
	dout2_6	AT %QX1.5:	BOOL;
	dout2_7	AT %QX1.6:	BOOL;
	su3_vent	AT %QX1.7:	BOOL;
	dout3_1	AT %QX2.0:	BOOL;
	spalnya_kontrazhur	AT %QX2.1:	BOOL; (*c*)
	spalnya_balkon				AT %QX2.2:	BOOL; (*c2*)
	dout3_4				AT %QX2.3:	BOOL;
	spalnya_kulbaba		AT %QX2.4:	BOOL;(*c3, c3a*)
	spalnya_kontrazhur_b	AT %QX2.5:	BOOL; (*c7*)
	spalnya_kontrazhur_l	AT %QX2.6:	BOOL; (*c4*)
	su3_stina			AT %QX2.7:	BOOL; (*c8*)
	(*dout4_1*)su3_pidsvitka 		AT %QX3.0:	BOOL;(*c10*)
	su3_bra				AT %QX3.1:	BOOL;(*c15*)
	su3_kontrazhur		AT %QX3.2:	BOOL;(*c9*)
	dytjacha				AT %QX3.3:	BOOL;(*c14*)
	su3_kontrazhur_k		AT %QX3.4:	BOOL; (*c11*)
	dytjacha_bra			AT %QX3.5:	BOOL; (*c15*)
	su3_lampa			AT %QX3.6:	BOOL; (*c12*)
	garderob			AT %QX3.7:	BOOL;
	(*dout5_1*)	serverna		AT %QX4.0:	BOOL;
	bar					AT %QX4.1:	BOOL;(*c21*)
	korydor_skeli 		AT %QX4.2:	BOOL;(*c18*)
	choven				AT %QX4.3:	BOOL;(*c22*)
	korydor_svitlo		AT %QX4.4:	BOOL;(*c19*)
	fancoil_spalnya_low 	AT %QX4.5:	BOOL;
	korydor_lampa		AT %QX4.6:	BOOL;(*c20*)
	fancoil_spalnya_med	AT %QX4.7:	BOOL;
	(*dout6_1*)fancoil_spalnya_high	AT%QX5.0:BOOL;
	rozetky1				AT%QX5.1 :BOOL;
	fancoil_dytjacha_low	AT%QX5.2 :BOOL;
	rozetky2			 	AT%QX5.3 :BOOL;
	fancoil_dytjacha_med	AT%QX5.4:BOOL;
	rozetky3 				AT%QX5.5:BOOL;
	fancoil_dytjacha_high	AT%QX5.6:BOOL;
	rozetky4 				AT%QX5.7:BOOL;
	(*dout7_1*)rozetky5	AT%QX6.0:BOOL;
	tul_close 			AT%QX6.1 :BOOL;
	rozetky6	 			AT%QX6.2 :BOOL;
	tul_open	 			AT%QX6.3 :BOOL;
	shtory_close 			AT%QX6.4:BOOL;
	lift_down				AT%QX6.5:BOOL;
	shtory_open			AT%QX6.6:BOOL;
	lift_up	 			AT%QX6.7:BOOL;
(*dout8_1*) dytjacha_col AT%QX7.0:BOOL; (*тепла підлога*)
	serverna_col 		AT%QX7.1 :BOOL;
	freshbar_col 			AT%QX7.2 :BOOL;
	spalnya_col 		AT%QX7.3 :BOOL;
	korydor_col		 	AT%QX7.4:BOOL;
	su_col_pidloga 		AT%QX7.5:BOOL;
	su_col_stina		AT%QX7.6:BOOL;
	out88 AT%QX7.7:BOOL;
	out91 AT%QX8.0:BOOL;
	out92 AT%QX8.1 :BOOL;
	out93 AT%QX8.2 :BOOL;
	out94 AT%QX8.3 :BOOL;
	out95 AT%QX8.4:BOOL;
	out96 AT%QX8.5:BOOL;
	out97 AT%QX8.6:BOOL;
	out98 AT%QX8.7:BOOL;

	klapan_dytjacha		AT %QB10:	INT;
	klapan_spalnya		AT %QB12:	INT;
	KL4414_3_Out		AT %QB14:	INT;
	klapan_vitalnya		AT %QB16:	INT;
(*light sensors*)
	iLight_N			AT %IB28:INT;
	iLight_W			AT %IB30:INT;
	iLight_S			AT %IB32:INT;
	iLight_E			AT %IB34:INT;

	KL6301_IN_0 AT %IB4: ARRAY[1..24] OF BYTE;
	KL6301_OUT_0 AT %QB34: ARRAY[1..24] OF BYTE;

	temp_tambur	AT %IB36: INT;(*тепла підлога*)
	temp_su		AT %IB38: INT;(*тепла підлога*)
	temp_spalnya	AT %IB40: INT;(*тепла підлога*)
	iT_out			AT %IB42:INT; (*зовнішня температура*)

END_VAR

(* Data type *)
TYPE ROOM_HVAC :
STRUCT
	manual_mode:BOOL;
	heat_mode: USINT; (*1-cool, 2-heat, 3-fan*)
	heat_speed: USINT;

	cur_t:REAL;
	cur_t_ust,cur_t_ust_prev, t_ust_heat,	t_ust_cool:REAL;
	cooling_signal,heating_signal:BYTE;

	fancoil_speed:SINT;
	klapan:WORD;

	tepla_pidloga:BOOL;

	zaslinka:BOOL;


END_STRUCT
END_TYPE

(* POU MAIN, ST *)
PROGRAM MAIN
VAR
	fbTimer: TON;
	fbRTC: RTC;
	i:INT;
	fbDarkTimeCorrection : TP;

	write1, write2, write4: BOOL;
	i2,j2,i1,j1, i4,j4: INT;
	repeat1, repeat2,repeat4:BOOL;


END_VAR
(*Parameters*)
	tLongPress:=t#500ms; (*затримка довгого натискання*)
	tOffDelay:=t#5m; (*затримка для відкладеного вимкнення*)

	ads_adr1:='10.0.5.61.1.1';
	ads_adr2:='10.0.5.62.1.1';
	ads_adr3:='10.0.5.63.1.1';
	ads_adr4:='10.0.5.64.1.1';

fbTimer(PT:=t#1s,IN:=NOT fbTimer.Q);

IF fbTimer.Q OR SYSTEMTASKINFOARR[1].firstCycle  THEN
	fbRTC;
END_IF


(*system_time:=DT_TO_SYSTEMTIME(fbRTC.CDT);*)
data1floor[4]:=WORD_TO_BYTE(system_time.wHour);
data1floor[5]:=WORD_TO_BYTE(system_time.wMinute);
data2floor[9]:=WORD_TO_BYTE(system_time.wHour);
data2floor[10]:=WORD_TO_BYTE(system_time.wMinute);
data_derevo[4]:=WORD_TO_BYTE(system_time.wHour);
data_derevo[5]:=WORD_TO_BYTE(system_time.wMinute);

fbDarkTimeCorrection(IN:=iLight_N<1000 AND  iLight_W <1000 AND iLight_S <1000 AND iLight_E <1000, PT:=t#40m);
IF iLight_N<1000 AND  iLight_W <1000 AND iLight_S <1000 AND iLight_E <1000  AND NOT fbDarkTimeCorrection.q AND ( system_time.wHour>15 OR system_time.wHour<9)  THEN
	bDarkOutside:=TRUE;
ELSE
	bDarkOutside:=FALSE;
END_IF



data2floor[6].1:=bDarkOutside;
data1floor[2].6:=bDarkOutside;
data_derevo[2].6:=bDarkOutside;

(*Світло*)
LIGHT;
shtory;

(*тепло*)
heat;

(*EIB init*)
EIB;

ADS_write;
ADS_Communication;
END_PROGRAM
ACTION ADS_write:
FOR i2:=0 TO (SIZEOF(data2floor))-1 DO
	IF data2floor[i2]<>data2floor_prev[i2]  THEN
		write2:=TRUE;
		EXIT;
	ELSE
		write2:=FALSE;
	END_IF
END_FOR


FOR i1:=0 TO (SIZEOF(data1floor))-1 DO
	IF data1floor[i1]<>data1floor_prev[i1]  THEN
		write1:=TRUE;
		EXIT;
	ELSE
		write1:=FALSE;
	END_IF
END_FOR


FOR i4:=0 TO (SIZEOF(data_derevo))-1 DO
	IF data_derevo[i4]<>data_derevo_prev[i4]  THEN
		write4:=TRUE;
		EXIT;
	ELSE
		write4:=FALSE;
	END_IF
END_FOR

FOR j1:=0 TO (SIZEOF(data1floor))-1 DO
	data1floor_prev[j1]:=data1floor[j1];
END_FOR

FOR j2:=0 TO (SIZEOF(data2floor))-1 DO
	data2floor_prev[j2]:=data2floor[j2];
END_FOR

FOR j4:=0 TO (SIZEOF(data_derevo))-1 DO
	data_derevo_prev[j4]:=data_derevo[j4];
END_FOR
END_ACTION

(* POU LIGHT, ST *)
PROGRAM LIGHT
VAR
	tambur1, tambur2,tambur3 : SWITCH;
	korydor : SWITCH;
	spalnya1,spalnya2, spalnya_balk:SWITCH;
	dytjacha1,dytjacha2  : SWITCH;
	su1 : SWITCH;
	su2: SWITCH;
	garderob1, garderob2 : SWITCH;

	tLightWindow: TIME;		(*Час, який світло світиться після спрацювання сенсора руху*)

	VENT_TIMER: TOF;		(*Таймер роботи вентилятора в пустому туалеті*)
	vent_timer_start: R_TRIG;
	test: BOOL;

	CHOVEN_TIMER: TOF;	(*Таймер роботи світильника на човні*)

	bChovenTimerOverride: SEMA;		(*Перевага вимикача над таймером*)
	bGarderobTimerOverride: SEMA;		(*Перевага вимикача над таймером*)
	KORYDOR_TIMER: TOF;		(*Таймер роботи світла в коридорі*)
	KORYDOR_F: F_TRIG;
	GARDEROB_TIMER: TOF;		(*Таймер роботи світла в гардеробі*)
	GARDEROB_F: F_TRIG;		(*Спрацювання сенсора руху в гардеробі*)
	KORYDOR_SEMA:SEMA;
	su_light: BOOL;
	vymykach3: BOOL;

	fb_light_write:EIB_BIT_SEND;
	block_korydor, block_garderob, block_choven: BOOL;

END_VAR
tLightWindow:=t#60s;

IF fb_moove_sensors_read.bData THEN
	moove_sensors:=(*bDarkOutside*)TRUE;
ELSE
	moove_sensors:=FALSE;
END_IF

(*Опитування вимикачів*)
tambur1(IN:=sw_tambur1);
tambur2(IN:=sw_tambur3_2);
tambur3(IN:=sw_tambur3);



spalnya1(IN:=sw_spalnya1 XOR sw_spalnya4);
spalnya2(IN:=sw_spalnya2 XOR sw_spalnya3);
spalnya_balk(IN:=sw_spalnya_balk);

dytjacha1(IN:=sw_dytjacha1);
dytjacha2(IN:=sw_dytjacha2);

su1(IN:=sw_su1);
su2(IN:=sw_su2);




(*запуск вечірніх таймерів світла*)





(*обробка сигналів вимикачів та таймерів*)
IF fb_bar_read.bDataReceive THEN
	IF tambur1.short THEN bar:= NOT bar; END_IF
ELSE
	bar:=fb_bar_read.bData;
END_IF

(*Відправка на 1,2 поверхи значення вимикача*)
data2floor[6].0:=sw_tambur3_2;
data1floor[2].1:=sw_tambur3_2;

CHOVEN_TIMER(IN:= NOT fb_choven_read.bData AND NOT moove_skhody, PT:= tLightWindow);
IF fb_choven_read.bData THEN
	choven:=TRUE;
ELSE
	IF moove_sensors  AND  CHOVEN_timer.Q	THEN  choven:=TRUE;
	ELSE
	choven:=FALSE;
	END_IF
END_IF


korydor(IN:=sw_korydor);
KORYDOR_TIMER(IN:=  NOT fb_korydor_lampa_read.bData  AND NOT moove_korydor, PT:= tLightWindow);

IF fb_korydor_lampa_read.bData THEN
	korydor_lampa:=TRUE;
ELSE
		korydor_lampa:=KORYDOR_TIMER.Q;
END_IF

IF fb_korydor_skeli_read.bData THEN
	korydor_skeli:=TRUE;
ELSE
	korydor_skeli:=KORYDOR_TIMER.Q;
END_IF

IF fb_korydor_svitlo_read.bDataReceive THEN
	KORYDOR_F(clk:=korydor_timer.Q);
	KORYDOR_SEMA(CLAIM:=(NOT korydor_svitlo AND korydor.short ), RELEASE:=(korydor_svitlo AND korydor.short) OR KORYDOR_f.Q);
	korydor_svitlo:=KORYDOR_SEMA.BUSY;
ELSE
	korydor_svitlo:= fb_korydor_svitlo_read.bData;

END_IF

IF fb_spalnya_kulbaba_read.bDataReceive THEN
	IF spalnya1.short THEN spalnya_kulbaba:=NOT spalnya_kulbaba; END_IF
ELSE
	spalnya_kulbaba:=fb_spalnya_kulbaba_read.bData;
END_IF

IF fb_spalnya_kontrazhur_read.bDataReceive XOR fb_spalnya_kontrazhur_b_read.bDataReceive  XOR fb_spalnya_kontrazhur_l_read.bDataReceive  THEN
	IF spalnya2.short THEN
		 spalnya_kontrazhur:= NOT spalnya_kontrazhur;
		spalnya_kontrazhur_b:=spalnya_kontrazhur;
		spalnya_kontrazhur_l:=spalnya_kontrazhur;
 	END_IF
ELSE
	IF NOT fb_spalnya_kontrazhur_read.bDataReceive THEN spalnya_kontrazhur:= fb_spalnya_kontrazhur_read.bData; END_IF
	IF NOT fb_spalnya_kontrazhur_l_read.bDataReceive THEN spalnya_kontrazhur_l:= fb_spalnya_kontrazhur_l_read.bData; END_IF
	IF NOT fb_spalnya_kontrazhur_b_read.bDataReceive THEN spalnya_kontrazhur_b:= fb_spalnya_kontrazhur_b_read.bData; END_IF
END_IF

IF fb_spalnya_balkon_read.bDataReceive THEN
	IF  spalnya_balk.short  THEN spalnya_balkon:=NOT spalnya_balkon; END_IF
ELSE
	spalnya_balkon:=fb_spalnya_balkon_read.bData;
END_IF

IF fb_dytjacha_read.bDataReceive THEN
	IF dytjacha1.short THEN dytjacha:= NOT dytjacha; END_IF
ELSE
	dytjacha:=fb_dytjacha_read.bData;
END_IF

IF fb_dytjacha_bra_read.bDataReceive THEN
	IF dytjacha2.short THEN dytjacha_bra:= NOT dytjacha_bra; END_IF
ELSE
	dytjacha_bra:=fb_dytjacha_bra_read.bData;
END_IF


IF fb_su3_stina_read.bDataReceive AND  fb_su3_kontrazhur_k_read.bDataReceive THEN
	IF su2.short THEN
		su3_stina:= NOT su3_stina;
		(*su3_kontrazhur_k:= su3_stina; *)
	END_IF
ELSE
	IF NOT fb_su3_stina_read.bDataReceive THEN
		 su3_stina:=fb_su3_stina_read.bData;
	END_IF
	IF NOT fb_su3_kontrazhur_k_read.bDataReceive THEN
		su3_kontrazhur_k:= fb_su3_kontrazhur_k_read.bData;
	END_IF
END_IF



IF fb_su3_bra_read.bDataReceive XOR fb_su3_lampa_read.bDataReceive XOR fb_su3_kontrazhur_read.bDataReceive THEN
	IF su2.long THEN
		su3_bra:= NOT su3_bra;
		su3_lampa:= su3_bra;
		su3_kontrazhur:=su3_lampa;
	END_IF
ELSE
	IF NOT  fb_su3_bra_read.bDataReceive THEN su3_bra:= fb_su3_bra_read.bData;END_IF
	IF NOT fb_su3_lampa_read.bDataReceive THEN su3_lampa:=fb_su3_lampa_read.bData; END_IF
	IF NOT  fb_su3_kontrazhur_read.bDataReceive THEN su3_kontrazhur:=fb_su3_kontrazhur_read.bData; END_IF
END_IF

IF su1.long THEN su3_vent:= NOT su3_vent; END_IF

IF fb_su3_pidsvitka_read.bDataReceive THEN
	IF su1.short THEN su3_pidsvitka:= NOT su3_pidsvitka; END_IF
ELSE
	su3_pidsvitka:=fb_su3_pidsvitka_read.bData;
END_IF

(*IF su1.short AND NOT su3_vent THEN su3_vent:=TRUE; END_IF; *) (*вмикання вентилятора разом зі світлом*)

(*
вмикання вентилятора на деякий час після того, як вимикається все світло у ванній

su_light:=su3_stina OR su3_kontrazhur OR su3_bra OR su3_pidsvitka;

vent_timer_start(CLK:=NOT su_light );
VENT_TIMER(PT:=tOffDelay,IN:=vent_timer_start.Q);
IF NOT su_light THEN
	su3_vent:= VENT_TIMER.Q;
END_IF
*)


garderob1(IN:=sw_garderob1);
garderob2(IN:=sw_garderob2);
GARDEROB_F(CLK:=moove_garderob);
GARDEROB_TIMER(IN:= GARDEROB_F.Q, PT:= tLightWindow*2);

IF fb_serverna_read.bDataReceive THEN
	IF garderob2.short THEN serverna := NOT serverna; END_IF
ELSE
	Serverna:=fb_serverna_read.bData;
END_IF

IF fb_garderob_read.bDataReceive THEN
(*	bGarderobTimerOverride(CLAIM:=  (NOT moove_garderob OR (NOT garderob AND garderob1.short)), RELEASE:=  (garderob AND  garderob1.short) );
	garderob:=bGarderobTimerOverride.BUSY;*)
	IF garderob1.short THEN garderob:= NOT garderob; END_IF
ELSE
	garderob:=fb_garderob_read.bData;
END_IF
END_PROGRAM

(* POU Vymykachi/SWITCH, ST *)
FUNCTION_BLOCK SWITCH
VAR_INPUT
	IN:BOOL;
	SHORT_OFF_DELAY, LONG_OFF_DELAY: TIME; (*час затримки вимкнення по короткому та довгому натисненню*)
END_VAR
VAR_OUTPUT
	short, long:BOOL;
END_VAR
VAR
	tChas: TIME; (*час доки кнопка натиснена*)
	TIMER: TON; (*таймер час натискання*)
	bPressed:BOOL;
	turn_off_long: BOOL;
	start_l, start_s:BOOL;
	bStan: BOOL:=FALSE;
END_VAR
short:=FALSE;
long:=FALSE;
TIMER(IN:=IN AND bStan, PT:=t#10s);
IF IN AND bStan THEN
	tChas:=timer.ET;
	bPressed:=TRUE;
ELSE
	bPressed:=FALSE;
END_IF;

IF NOT IN AND NOT bStan THEN
	tChas:=t#0ms;
END_IF;

IF bStan AND NOT IN THEN
	IF tChas <tLongPress THEN
		short:=TRUE;
	END_IF;
	IF tChas>=tLongPress THEN
		long:=TRUE;
	END_IF;
END_IF;
bStan := IN;
END_FUNCTION_BLOCK

(* POU shtory, ST *)
PROGRAM shtory
VAR
	inc1, inc: UINT;
	impulse: BOOL;
	last_move: UINT;
	impulse1: BOOL;
	last_move1: UINT;
	lift_move_dir, lift_move: BOOL;
	rising1: BOOL;
	falling1: BOOL;
	rising2: BOOL;
	falling2: BOOL;
	panel_shtory_move, panel_tul_move, panel_lift_move:BOOL;

	(*таймери для формування керуючих імпульсів*)
	timer_shtory_move, timer_shtory_stop,timer_tul_move, timer_tul_stop, move_lift_up, move_lift_down: TP;
	counter:CTU;
	shtory_move: BOOL;
	tul_move: BOOL;
	bBlock:BOOL;
	darkness_shtory_move: TP;
	btest: BOOL;

	eib_spalnya_shtory_status_send: EIB_BIT_SEND;
	eib_spalnya_tul_status_send: EIB_BIT_SEND;
	spalnya_shtory_status: BOOL;
	spalnya_tul_status: BOOL;
END_VAR
bBlock:=FALSE;
IF MAIN.fbRTC.stSystemTime.wHour=11 AND MAIN.fbRTC.stSystemTime.wMinute=0 AND MAIN.fbRTC.stSystemTime.wSecond<22 THEN
	bBlock:=TRUE;
	lift_down:=TRUE;
	lift_up:=FALSE;
	lift_move_dir:=FALSE;
	shtory_open:=TRUE;
	shtory_close:=FALSE;
	tul_open:=FALSE;
	tul_close:=TRUE;

ELSE
	(*детекція відсутності фронтів*)
	IF LIGHT.spalnya1.long = impulse THEN
		rising1:=0;
		falling1:=0;
	END_IF;

	IF LIGHT.spalnya2.long = impulse1  THEN
		rising2:=0;
		falling2:=0;
	END_IF;

	(*якщо клавіші довго  натиснені одночасно, то рухати ліфт, якщо довго і окремо - штори*)
	IF ( (LIGHT.spalnya1.long AND LIGHT.spalnya2.long) OR panel_lift_move)  AND NOT( move_lift_up.Q OR  move_lift_down.Q)  THEN
		lift_move:=1;
		lift_move_dir:= NOT lift_move_dir;
	ELSE

		(*ловим передній фронт довгого натискання першої клавіші*)
		IF LIGHT.spalnya1.long AND NOT impulse  AND NOT LIGHT.spalnya2.long THEN
			rising1:=1;
			falling1:=0;
		END_IF;

		(*задній фронт*)
		IF NOT LIGHT.spalnya1.long AND  impulse AND NOT LIGHT.spalnya2.long  THEN
			falling1:=1;
			rising1:=0;
		END_IF;

		(*ловим передній фронт довгого натискання другої клавіші*)
		IF LIGHT.spalnya2.long AND NOT impulse1 AND NOT LIGHT.spalnya1.long  THEN
			rising2:=1;
			falling2:=0;
		END_IF;

		(*ловим задній фронт довгого натискання другої клавіші*)
		IF NOT LIGHT.spalnya2.long AND  impulse1 AND NOT LIGHT.spalnya1.long THEN
			falling2:=1;
			rising2:=0;
		END_IF
	END_IF
	(*команди шторам та ліфту з панелей смартбаса*)
	eib_shtory(Group_Address:=shtory_spalnya_EIB_addr, strData_Rec:=fb_KL6301_0.str_Data_Rec);
	eib_tul(Group_Address:=tul_spalnya_EIB_addr, strData_Rec:=fb_KL6301_0.str_Data_Rec);
	eib_lift(Group_Address:=lift_spalnya_EIB_addr, strData_Rec:=fb_KL6301_0.str_Data_Rec);


	IF NOT eib_shtory_kabinet.bDataReceive THEN data2floor[7].0:=eib_shtory_kabinet.bData; END_IF
	IF NOT eib_tul_kabinet.bDataReceive THEN data2floor[7].1:=eib_tul_kabinet.bData; END_IF
	IF NOT eib_shtory_kino.bDataReceive THEN data2floor[7].2:=eib_shtory_kino.bData; END_IF
	IF NOT eib_tul_kino.bDataReceive THEN data2floor[7].3:=eib_tul_kino.bData; END_IF

	panel_tul_move:= NOT eib_tul.bDataReceive;
	panel_shtory_move:= NOT eib_shtory.bDataReceive;
	panel_lift_move:=NOT eib_lift.bDataReceive;


	shtory_move:= LIGHT.spalnya1.long OR panel_shtory_move;
	tul_move:= LIGHT.spalnya2.long OR panel_tul_move;



	(*формування імпульсів для керування шторами, тюлями та ліфтом*)
	timer_shtory_move(IN:=shtory_move, PT:=t#500ms);
	timer_shtory_stop(IN:=shtory_move , PT:=t#500ms);
	timer_tul_move(IN:=tul_move  , PT:=t#500ms);
	timer_tul_stop(IN:=tul_move , PT:=t#500ms);

	move_lift_up(IN:=lift_move AND lift_move_dir , PT:=t#20s,Q=>lift_up);
	move_lift_down(IN:=lift_move AND NOT lift_move_dir, PT:=t#20s, Q=>lift_down);



	darkness_shtory_move(IN:=bDarkOutside, PT:=t#15s);
	IF darkness_shtory_move.Q THEN
		shtory_open:=FALSE;
		shtory_close:=TRUE;
		tul_open:=FALSE;
		tul_close:=TRUE;
		bBlock:=TRUE;
	END_IF


	IF NOT bBlock THEN
		IF NOT (LIGHT.spalnya1.long AND LIGHT.spalnya2.long) THEN (*якщо не засік довгого затискання двох клавіш (ліфт не рухається) - рухати штори *)

		(*вибір рухати чи зупинити  штори*)
			IF shtory_move   THEN
				inc:=inc+1;
			END_IF;
			IF inc>2 THEN inc:=1; END_IF;

			(*вибір рухати чи зупинити  тюль*)
			IF tul_move THEN
				inc1:=inc1+1;
			END_IF;
			IF inc1>2 THEN inc1:=1; END_IF;

			CASE inc OF

				1:
				shtory_open:=timer_shtory_move.Q; (*відкривати*)
				shtory_close:= 0;
				last_move:=inc;
				spalnya_shtory_status:=1;

				2:
				shtory_close:=timer_shtory_move.Q;(*закривати*)
				shtory_open:= 0;
				last_move:=inc;
				spalnya_shtory_status:=0;

			END_CASE;

			CASE inc1 OF

				1:
				tul_open:=timer_tul_move.Q; (*відкривати*)
				tul_close:= 0;
				last_move1:=inc;
				spalnya_tul_status:=1;
				2:
				tul_close:=timer_tul_move.Q;(*закривати*)
				tul_open:= 0;
				last_move1:=inc;
				spalnya_tul_status:=0;
			END_CASE;

		END_IF;
	END_IF

	(*запам'ятовування стану довгого натискання для детекції фронтів*)

	impulse:=LIGHT.spalnya1.long;
	impulse1:=LIGHT.spalnya2.long;

	 lift_move:= 0;
END_IF
eib_status_send;

new_shtory;
END_PROGRAM
ACTION eib_status_send:
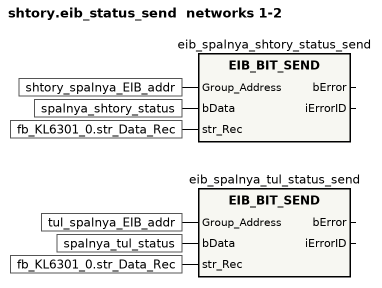
_FBD_ (* Function Block Diagram *)
NETWORK 1
	eib_spalnya_shtory_status_send:EIB_BIT_SEND(Group_Address: shtory_spalnya_EIB_addr, bData: spalnya_shtory_status, str_Rec: fb_KL6301_0.str_Data_Rec)
NETWORK 2
	eib_spalnya_tul_status_send:EIB_BIT_SEND(Group_Address: tul_spalnya_EIB_addr, bData: spalnya_tul_status, str_Rec: fb_KL6301_0.str_Data_Rec)
_END_FBD_
(* the same logic as Structured Text *)
(* Network 1 *)
eib_spalnya_shtory_status_send(Group_Address := shtory_spalnya_EIB_addr, bData := spalnya_shtory_status, str_Rec := fb_KL6301_0.str_Data_Rec);
(* Network 2 *)
eib_spalnya_tul_status_send(Group_Address := tul_spalnya_EIB_addr, bData := spalnya_tul_status, str_Rec := fb_KL6301_0.str_Data_Rec);
END_ACTION

(* POU new_shtory, CFC *)
PROGRAM new_shtory
VAR

END_VAR
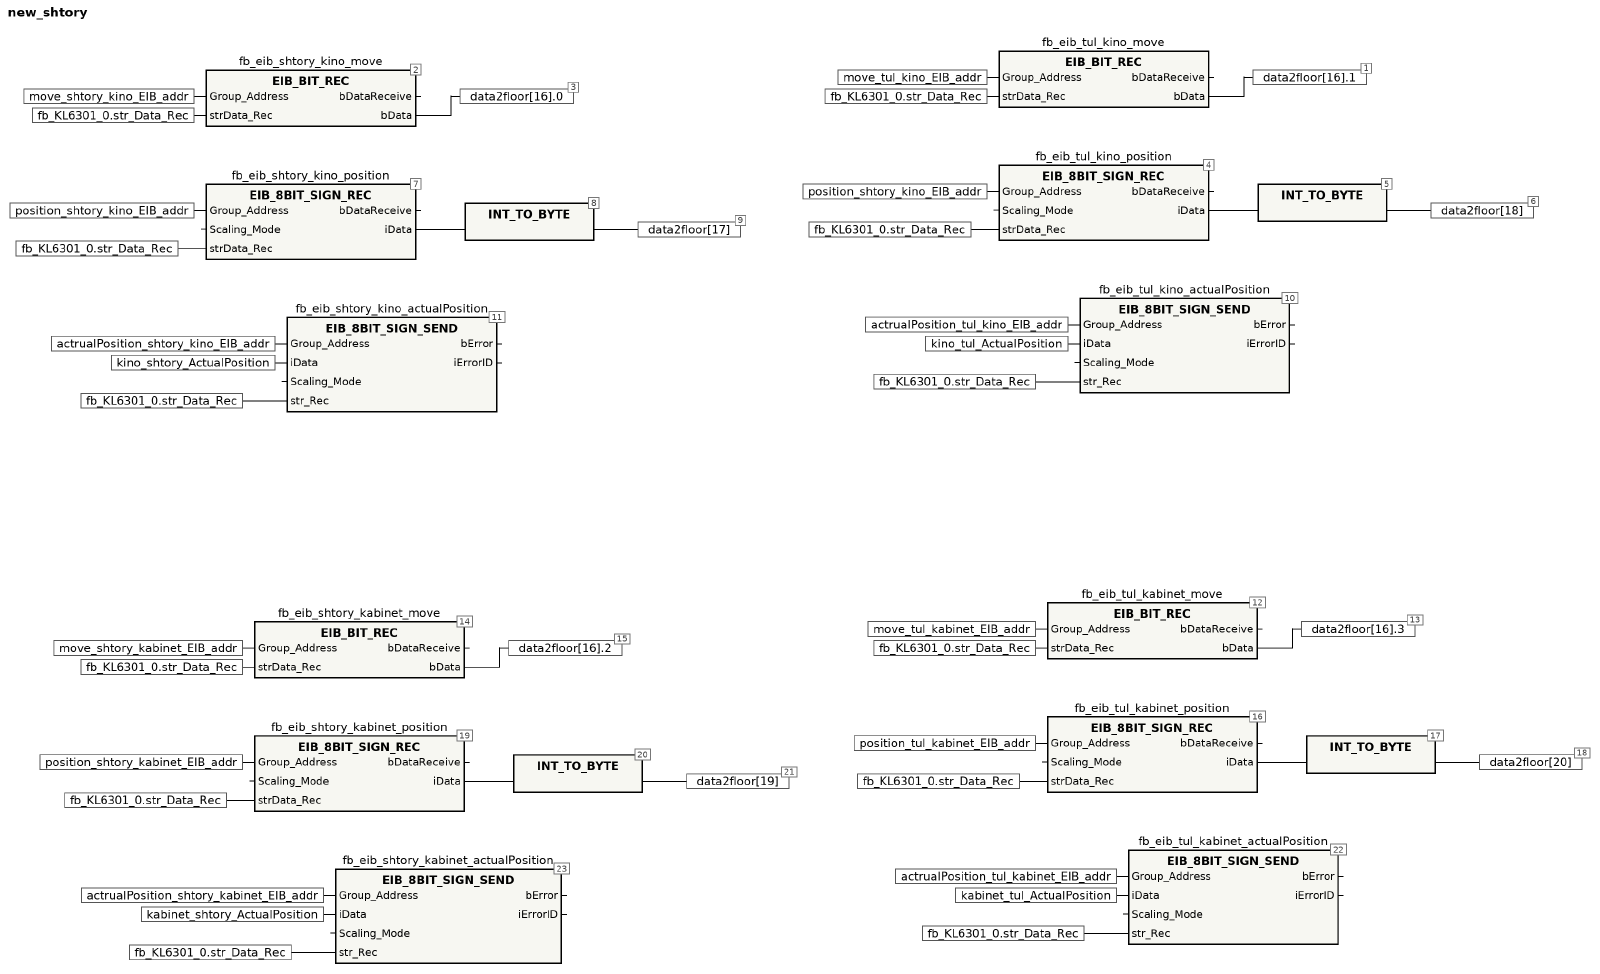
_CFC_ (* Continuous Function Chart, elements in execution order *)
#0 fb_eib_tul_kino_move:EIB_BIT_REC(Group_Address: move_tul_kino_EIB_addr, strData_Rec: fb_KL6301_0.str_Data_Rec)
#1 data2floor[16].1 <= #0.bData
#2 fb_eib_shtory_kino_move:EIB_BIT_REC(Group_Address: move_shtory_kino_EIB_addr, strData_Rec: fb_KL6301_0.str_Data_Rec)
#3 data2floor[16].0 <= #2.bData
#4 fb_eib_tul_kino_position:EIB_8BIT_SIGN_REC(Group_Address: position_shtory_kino_EIB_addr, Scaling_Mode: -, strData_Rec: fb_KL6301_0.str_Data_Rec)
#5 INT_TO_BYTE(#4.iData)
#6 data2floor[18] <= #5
#7 fb_eib_shtory_kino_position:EIB_8BIT_SIGN_REC(Group_Address: position_shtory_kino_EIB_addr, Scaling_Mode: -, strData_Rec: fb_KL6301_0.str_Data_Rec)
#8 INT_TO_BYTE(#7.iData)
#9 data2floor[17] <= #8
#10 fb_eib_tul_kino_actualPosition:EIB_8BIT_SIGN_SEND(Group_Address: actrualPosition_tul_kino_EIB_addr, iData: kino_tul_ActualPosition, Scaling_Mode: -, str_Rec: fb_KL6301_0.str_Data_Rec)
#11 fb_eib_shtory_kino_actualPosition:EIB_8BIT_SIGN_SEND(Group_Address: actrualPosition_shtory_kino_EIB_addr, iData: kino_shtory_ActualPosition, Scaling_Mode: -, str_Rec: fb_KL6301_0.str_Data_Rec)
#12 fb_eib_tul_kabinet_move:EIB_BIT_REC(Group_Address: move_tul_kabinet_EIB_addr, strData_Rec: fb_KL6301_0.str_Data_Rec)
#13 data2floor[16].3 <= #12.bData
#14 fb_eib_shtory_kabinet_move:EIB_BIT_REC(Group_Address: move_shtory_kabinet_EIB_addr, strData_Rec: fb_KL6301_0.str_Data_Rec)
#15 data2floor[16].2 <= #14.bData
#16 fb_eib_tul_kabinet_position:EIB_8BIT_SIGN_REC(Group_Address: position_tul_kabinet_EIB_addr, Scaling_Mode: -, strData_Rec: fb_KL6301_0.str_Data_Rec)
#17 INT_TO_BYTE(#16.iData)
#18 data2floor[20] <= #17
#19 fb_eib_shtory_kabinet_position:EIB_8BIT_SIGN_REC(Group_Address: position_shtory_kabinet_EIB_addr, Scaling_Mode: -, strData_Rec: fb_KL6301_0.str_Data_Rec)
#20 INT_TO_BYTE(#19.iData)
#21 data2floor[19] <= #20
#22 fb_eib_tul_kabinet_actualPosition:EIB_8BIT_SIGN_SEND(Group_Address: actrualPosition_tul_kabinet_EIB_addr, iData: kabinet_tul_ActualPosition, Scaling_Mode: -, str_Rec: fb_KL6301_0.str_Data_Rec)
#23 fb_eib_shtory_kabinet_actualPosition:EIB_8BIT_SIGN_SEND(Group_Address: actrualPosition_shtory_kabinet_EIB_addr, iData: kabinet_shtory_ActualPosition, Scaling_Mode: -, str_Rec: fb_KL6301_0.str_Data_Rec)
_END_CFC_
(* the same logic as Structured Text *)
fb_eib_tul_kino_move(Group_Address := move_tul_kino_EIB_addr, strData_Rec := fb_KL6301_0.str_Data_Rec);
data2floor[16].1 := fb_eib_tul_kino_move.bData;
fb_eib_shtory_kino_move(Group_Address := move_shtory_kino_EIB_addr, strData_Rec := fb_KL6301_0.str_Data_Rec);
data2floor[16].0 := fb_eib_shtory_kino_move.bData;
fb_eib_tul_kino_position(Group_Address := position_shtory_kino_EIB_addr, strData_Rec := fb_KL6301_0.str_Data_Rec);
data2floor[18] := INT_TO_BYTE(fb_eib_tul_kino_position.iData);
fb_eib_shtory_kino_position(Group_Address := position_shtory_kino_EIB_addr, strData_Rec := fb_KL6301_0.str_Data_Rec);
data2floor[17] := INT_TO_BYTE(fb_eib_shtory_kino_position.iData);
fb_eib_tul_kino_actualPosition(Group_Address := actrualPosition_tul_kino_EIB_addr, iData := kino_tul_ActualPosition, str_Rec := fb_KL6301_0.str_Data_Rec);
fb_eib_shtory_kino_actualPosition(Group_Address := actrualPosition_shtory_kino_EIB_addr, iData := kino_shtory_ActualPosition, str_Rec := fb_KL6301_0.str_Data_Rec);
fb_eib_tul_kabinet_move(Group_Address := move_tul_kabinet_EIB_addr, strData_Rec := fb_KL6301_0.str_Data_Rec);
data2floor[16].3 := fb_eib_tul_kabinet_move.bData;
fb_eib_shtory_kabinet_move(Group_Address := move_shtory_kabinet_EIB_addr, strData_Rec := fb_KL6301_0.str_Data_Rec);
data2floor[16].2 := fb_eib_shtory_kabinet_move.bData;
fb_eib_tul_kabinet_position(Group_Address := position_tul_kabinet_EIB_addr, strData_Rec := fb_KL6301_0.str_Data_Rec);
data2floor[20] := INT_TO_BYTE(fb_eib_tul_kabinet_position.iData);
fb_eib_shtory_kabinet_position(Group_Address := position_shtory_kabinet_EIB_addr, strData_Rec := fb_KL6301_0.str_Data_Rec);
data2floor[19] := INT_TO_BYTE(fb_eib_shtory_kabinet_position.iData);
fb_eib_tul_kabinet_actualPosition(Group_Address := actrualPosition_tul_kabinet_EIB_addr, iData := kabinet_tul_ActualPosition, str_Rec := fb_KL6301_0.str_Data_Rec);
fb_eib_shtory_kabinet_actualPosition(Group_Address := actrualPosition_shtory_kabinet_EIB_addr, iData := kabinet_shtory_ActualPosition, str_Rec := fb_KL6301_0.str_Data_Rec);
END_PROGRAM

(* POU HVAC/heat, ST *)
PROGRAM heat
VAR PERSISTENT

	t_out, t_out_avg_day, t_out_avg_10day:REAL;
	measures_this_day, meashured_days:INT;
	day_sum, ten_day_sum:REAL;
END_VAR


VAR
	temp_measure:TOF; (*таймер задає частоту замірів температури*)
	(*актуальна та попередня температури*)
	t_tambur, t_tamburPrev: REAL;
	t_su, t_suPrev: REAL;
	t_spalnya, t_spalnyaPrev: REAL;
	t_outPrev:REAL;
	(*мінімум та максимум температур теплих підлог*)
	t_max: REAL;
	t_min: REAL;
	(*різниця між поперднім та актуальним значенням температури*)
	delta_out, delta_tambur, delta_su, delta_spalnya: REAL;

	i: INT:=0;
	fbRetryCounter:CTU;
	iRetryCounter:INT;
	(*використовуються для знаходження середньої температури при ініціації*)
	t_tambur_sum: REAL;
	t_su_sum: REAL;
	t_spalnya_sum: REAL;
	t_out_sum: REAL;
	retry: BOOL:=TRUE;		(*переміряти температуру*)
END_VAR
(*фільтр показань сенсорів температури*)
CASE i OF
0..500: init;
ELSE
	IF retry THEN
		temp_measure.PT:=t#2s;

	ELSE temp_measure.PT:=t#5m;
	END_IF
	IF retry THEN
		IF iRetryCounter >5 THEN iRetryCounter:=0; i:=0; ELSE iRetryCounter:=iRetryCounter+1; END_IF;
	END_IF;
	temp_measure( IN:=NOT temp_measure.q); (*перевіряти температуру кожні 20 хв*)


IF NOT temp_measure.Q THEN

	delta_spalnya:=ABS(t_spalnyaPrev-temp_spalnya*0.1);
	delta_su:=ABS(t_suPrev-temp_su*0.1);
	delta_tambur:=ABS(t_tamburPrev-temp_tambur*0.1);
	delta_out:=ABS(t_outPrev-iT_out*0.1);
	retry:=FALSE;
	IF delta_spalnya<1 THEN
		t_spalnya:= temp_spalnya * 0.1;
	ELSE
		t_spalnya:=t_spalnyaPrev;
		retry:=TRUE;
	END_IF

	IF delta_su<1 THEN
		t_su:= temp_su * 0.1;
	ELSE
		t_su:=t_suPrev;
		retry:=TRUE;
	END_IF

	IF delta_tambur<1 THEN
		t_tambur:= temp_tambur * 0.1;
	ELSE
		t_tambur:=t_tamburPrev;
		retry:=TRUE;
	END_IF

	IF delta_out<01 THEN
		t_out:= iT_out* 0.1;
	ELSE
		t_out:=t_outPrev;
		retry:=TRUE;
	END_IF

	t_spalnyaPrev:=t_spalnya;
	t_suPrev:=t_su;
	t_tamburPrev:=t_tambur;
	t_outPrev:=t_out;

END_IF
END_CASE

(*CASE MAIN.fbRTC.stSystemTime.wSecond OF*)

IF t_out<0 THEN data1floor[2].7:=1; ELSE data1floor[2].7:=0; END_IF
data1floor[3]:=ABS(REAL_TO_BYTE(t_out));
data2floor[8]:=ABS(REAL_TO_BYTE(t_out));

(*summer; *)

t_max:=70;
t_min:=20;
IF t_out<15 THEN

	IF t_tambur > t_max THEN (*вимкнути колектор, якщо підлога тепліша за верхню межу температури*)
		freshbar_col:=FALSE;
	ELSE
		IF t_tambur< t_min THEN (*увімкнути колектор, якщо підлога холодніша за нижню межу*)
			freshbar_col:=TRUE;
		ELSE
			freshbar_col:= FALSE; (*ПОСТАВИТИ В ЗАЛЕЖНІСТЬ ВІД ЗОВНІШНЬОЇ ТЕМПЕРАТУРИ*)
		END_IF
	END_IF

	IF t_su > t_max THEN
		su_col_pidloga:=FALSE;
		su_col_stina:=FALSE;
			serverna_col:=FALSE;
	ELSE
		IF t_su< t_min THEN
			su_col_pidloga:=TRUE;
			su_col_stina:=TRUE;
			serverna_col:=TRUE;
		ELSE
			su_col_pidloga:=FALSE; (*ПОСТАВИТИ В ЗАЛЕЖНІСТЬ ВІД ЗОВНІШНЬОЇ ТЕМПЕРАТУРИ*)
			su_col_stina:=FALSE;
			serverna_col:=FALSE;
		END_IF
	END_IF

	IF t_spalnya>t_max THEN (*щоб не вистигала підлога*)
		spalnya_col:=FALSE;
	ELSE
		IF t_spalnya<t_min THEN
			spalnya_col:=TRUE;
		ELSE
			spalnya_col:=SPALNYA_HVAC.tepla_pidloga;
		END_IF
	END_IF


END_IF

(*

IF VITALNYA_HVAC.heat_mode=0 THEN
				VITALNYA_HVAC.fancoil_speed:=0;
				(*VITALNYA_HVAC.collector:=2#00000000; all closed*)
				VITALNYA_HVAC.klapan:=16#7FFF;(*full closed*)
				VITALNYA_HVAC.zaslinka:=TRUE;(*closed*)
	END_IF

	IF KINO_HVAC.heat_mode=0 THEN
				KINO_HVAC.fancoil_speed:=0;
				(*KINO_HVAC.collector:=2#00000000; all closed*)
				KINO_HVAC.klapan:=16#7FFF;(*full closed*)
				KINO_HVAC.zaslinka:=TRUE;(*closed*)
	END_IF

	IF STUDIO_HVAC.heat_mode=0 THEN
				STUDIO_HVAC.fancoil_speed:=0;
				(*STUDIO_HVAC.collector:=2#00000000; all closed*)
				STUDIO_HVAC.klapan:=16#7FFF;(*full closed*)
				STUDIO_HVAC.zaslinka:=TRUE;(*closed*)
	END_IF

	IF KABINET_HVAC.heat_mode=0 THEN
				KABINET_HVAC.fancoil_speed:=0;
				(*KABINET_HVAC.collector:=2#00000000; all closed*)
				KABINET_HVAC.klapan:=16#7FFF;(*full closed*)
				KABINET_HVAC.zaslinka:=TRUE;(*closed*)
	END_IF

	IF DYTJACHA_HVAC.heat_mode=0 THEN
				DYTJACHA_HVAC.fancoil_speed:=0;
				(*DYTJACHA_HVAC.collector:=2#00000000; all closed*)
				DYTJACHA_HVAC.klapan:=16#7FFF;(*full closed*)
				DYTJACHA_HVAC.zaslinka:=TRUE;(*closed*)
	END_IF

	IF SPALNYA_HVAC.heat_mode=0 THEN
				SPALNYA_HVAC.fancoil_speed:=0;
				(*SPALNYA_HVAC.collector:=2#00000000; all closed*)
				SPALNYA_HVAC.klapan:=16#7FFF;(*full closed*)
				SPALNYA_HVAC.zaslinka:=TRUE;(*closed*)
	END_IF
*)


data1floor[3]:=REAL_TO_BYTE (t_out);
data2floor[8]:=REAL_TO_BYTE (t_out);
data_derevo[3]:=REAL_TO_BYTE (t_out);
(*локальні змінні для фенкойлів 3го поверхну об'явлені в області виходів*)

(*------------------------fancoil speed --------------------------------------------------*)
IF EIB.fb_vitalnya_damper_ctrl_rec.bData THEN
	vitalnya_hvac.fancoil_speed:=1;
ELSE
	IF vitalnya_HVAC.heating_signal = 0  THEN
		CASE vitalnya_hvac.fancoil_speed OF
			0:	IF vitalnya_hvac.cooling_signal>0 THEN vitalnya_HVAC.fancoil_speed:=1; END_IF

			1:	IF vitalnya_hvac.cooling_signal=0 THEN vitalnya_HVAC.fancoil_speed:=0; END_IF
				IF vitalnya_hvac.cooling_signal>50 THEN  vitalnya_HVAC.fancoil_speed:=2; END_IF

			2:	IF vitalnya_hvac.cooling_signal=0 THEN vitalnya_HVAC.fancoil_speed:=0; END_IF
				IF vitalnya_hvac.cooling_signal>75  THEN vitalnya_HVAC.fancoil_speed:=3; END_IF
				IF vitalnya_hvac.cooling_signal<45  THEN vitalnya_HVAC.fancoil_speed:=1; END_IF

			3:	IF vitalnya_hvac.cooling_signal=0 THEN vitalnya_HVAC.fancoil_speed:=0; END_IF
				IF vitalnya_hvac.cooling_signal<75  THEN vitalnya_HVAC.fancoil_speed:=2; END_IF
		END_CASE
	END_IF

	IF vitalnya_HVAC.cooling_signal = 0 THEN
		CASE vitalnya_hvac.fancoil_speed OF
			0:	IF vitalnya_hvac.heating_signal>0 THEN vitalnya_HVAC.fancoil_speed:=1; END_IF

			1:	IF vitalnya_hvac.heating_signal=0 THEN vitalnya_HVAC.fancoil_speed:=0; END_IF
				IF vitalnya_hvac.heating_signal>50 THEN  vitalnya_HVAC.fancoil_speed:=2; END_IF

			2:	IF vitalnya_hvac.heating_signal=0 THEN vitalnya_HVAC.fancoil_speed:=0; END_IF
				IF vitalnya_hvac.heating_signal>75  THEN vitalnya_HVAC.fancoil_speed:=3; END_IF
				IF vitalnya_hvac.heating_signal<45  THEN vitalnya_HVAC.fancoil_speed:=1; END_IF

			3:	IF vitalnya_hvac.heating_signal=0 THEN vitalnya_HVAC.fancoil_speed:=0; END_IF
				IF vitalnya_hvac.heating_signal<75  THEN vitalnya_HVAC.fancoil_speed:=2; END_IF
		END_CASE
	END_IF
END_IF

IF EIB.fb_kino_damper_ctrl_rec.bData THEN
	kino_hvac.fancoil_speed:=1;
ELSE
	IF kino_HVAC.heating_signal = 0 THEN
		CASE kino_hvac.fancoil_speed OF
			0:	IF kino_hvac.cooling_signal>0 THEN kino_HVAC.fancoil_speed:=1; END_IF

			1:	IF kino_hvac.cooling_signal=0 THEN kino_HVAC.fancoil_speed:=0; END_IF
				IF kino_hvac.cooling_signal>50 THEN  kino_HVAC.fancoil_speed:=2; END_IF

			2:	IF kino_hvac.cooling_signal=0 THEN kino_HVAC.fancoil_speed:=0; END_IF
				IF kino_hvac.cooling_signal>75  THEN kino_HVAC.fancoil_speed:=3; END_IF
				IF kino_hvac.cooling_signal<45  THEN kino_HVAC.fancoil_speed:=1; END_IF

			3:	IF kino_hvac.cooling_signal=0 THEN kino_HVAC.fancoil_speed:=0; END_IF
				IF kino_hvac.cooling_signal<75  THEN kino_HVAC.fancoil_speed:=2; END_IF
		END_CASE
	END_IF
	IF kino_HVAC.cooling_signal = 0 THEN
		CASE kino_hvac.fancoil_speed OF
			0:	IF kino_hvac.heating_signal>0 THEN kino_HVAC.fancoil_speed:=1; END_IF

			1:	IF kino_hvac.heating_signal=0 THEN kino_HVAC.fancoil_speed:=0; END_IF
				IF kino_hvac.heating_signal>50 THEN  kino_HVAC.fancoil_speed:=2; END_IF

			2:	IF kino_hvac.heating_signal=0 THEN kino_HVAC.fancoil_speed:=0; END_IF
				IF kino_hvac.heating_signal>75  THEN kino_HVAC.fancoil_speed:=3; END_IF
				IF kino_hvac.heating_signal<45  THEN kino_HVAC.fancoil_speed:=1; END_IF

			3:	IF kino_hvac.heating_signal=0 THEN kino_HVAC.fancoil_speed:=0; END_IF
				IF kino_hvac.heating_signal<75  THEN kino_HVAC.fancoil_speed:=2; END_IF
		END_CASE
	END_IF
END_IF

IF EIB.fb_kabinet_damper_ctrl_rec.bData THEN
	kabinet_hvac.fancoil_speed:=1;
ELSE
	IF kabinet_HVAC.heating_signal = 0 THEN
		CASE kabinet_hvac.fancoil_speed OF
			0:	IF kabinet_hvac.cooling_signal>0 THEN kabinet_HVAC.fancoil_speed:=1; END_IF

			1:	IF kabinet_hvac.cooling_signal=0 THEN kabinet_HVAC.fancoil_speed:=0; END_IF
				IF kabinet_hvac.cooling_signal>50 THEN  kabinet_HVAC.fancoil_speed:=2; END_IF

			2:	IF kabinet_hvac.cooling_signal=0 THEN kabinet_HVAC.fancoil_speed:=0; END_IF
				IF kabinet_hvac.cooling_signal>75  THEN kabinet_HVAC.fancoil_speed:=3; END_IF
				IF kabinet_hvac.cooling_signal<45  THEN kabinet_HVAC.fancoil_speed:=1; END_IF

			3:	IF kabinet_hvac.cooling_signal=0 THEN kabinet_HVAC.fancoil_speed:=0; END_IF
				IF kabinet_hvac.cooling_signal<75  THEN kabinet_HVAC.fancoil_speed:=2; END_IF
		END_CASE
	END_IF
	IF kabinet_HVAC.cooling_signal = 0 THEN
		CASE kabinet_hvac.fancoil_speed OF
			0:	IF kabinet_hvac.heating_signal>0 THEN kabinet_HVAC.fancoil_speed:=1; END_IF

			1:	IF kabinet_hvac.heating_signal=0 THEN kabinet_HVAC.fancoil_speed:=0; END_IF
				IF kabinet_hvac.heating_signal>50 THEN  kabinet_HVAC.fancoil_speed:=2; END_IF

			2:	IF kabinet_hvac.heating_signal=0 THEN kabinet_HVAC.fancoil_speed:=0; END_IF
				IF kabinet_hvac.heating_signal>75  THEN kabinet_HVAC.fancoil_speed:=3; END_IF
				IF kabinet_hvac.heating_signal<45  THEN kabinet_HVAC.fancoil_speed:=1; END_IF

			3:	IF kabinet_hvac.heating_signal=0 THEN kabinet_HVAC.fancoil_speed:=0; END_IF
				IF kabinet_hvac.heating_signal<75  THEN kabinet_HVAC.fancoil_speed:=2; END_IF
		END_CASE
	END_IF
END_IF

IF EIB.fb_dytjacha_damper_ctrl_rec.bData THEN
	dytjacha_hvac.fancoil_speed:=1;
ELSE
	IF dytjacha_HVAC.heating_signal = 0 THEN
		CASE dytjacha_hvac.fancoil_speed OF
			0:	IF dytjacha_hvac.cooling_signal>0 THEN dytjacha_HVAC.fancoil_speed:=1; END_IF

			1:	IF dytjacha_hvac.cooling_signal=0 THEN dytjacha_HVAC.fancoil_speed:=0; END_IF
				IF dytjacha_hvac.cooling_signal>50 THEN  dytjacha_HVAC.fancoil_speed:=2; END_IF

			2:	IF dytjacha_hvac.cooling_signal=0 THEN dytjacha_HVAC.fancoil_speed:=0; END_IF
				IF dytjacha_hvac.cooling_signal>75  THEN dytjacha_HVAC.fancoil_speed:=3; END_IF
				IF dytjacha_hvac.cooling_signal<45  THEN dytjacha_HVAC.fancoil_speed:=1; END_IF

			3:	IF dytjacha_hvac.cooling_signal=0 THEN dytjacha_HVAC.fancoil_speed:=0; END_IF
				IF dytjacha_hvac.cooling_signal<75  THEN dytjacha_HVAC.fancoil_speed:=2; END_IF
		END_CASE
	END_IF
	IF dytjacha_HVAC.cooling_signal = 0 THEN
		CASE dytjacha_hvac.fancoil_speed OF
			0:	IF dytjacha_hvac.heating_signal>0 THEN dytjacha_HVAC.fancoil_speed:=1; END_IF

			1:	IF dytjacha_hvac.heating_signal=0 THEN dytjacha_HVAC.fancoil_speed:=0; END_IF
				IF dytjacha_hvac.heating_signal>50 THEN  dytjacha_HVAC.fancoil_speed:=2; END_IF

			2:	IF dytjacha_hvac.heating_signal=0 THEN dytjacha_HVAC.fancoil_speed:=0; END_IF
				IF dytjacha_hvac.heating_signal>75  THEN dytjacha_HVAC.fancoil_speed:=3; END_IF
				IF dytjacha_hvac.heating_signal<45  THEN dytjacha_HVAC.fancoil_speed:=1; END_IF

			3:	IF dytjacha_hvac.heating_signal=0 THEN dytjacha_HVAC.fancoil_speed:=0; END_IF
				IF dytjacha_hvac.heating_signal<75  THEN dytjacha_HVAC.fancoil_speed:=2; END_IF
		END_CASE
	END_IF
END_IF

IF EIB.fb_spalnya_damper_ctrl_rec.bData THEN
	spalnya_hvac.fancoil_speed:=1;
ELSE
	IF spalnya_HVAC.heating_signal = 0 THEN
		CASE spalnya_hvac.fancoil_speed OF
			0:	IF spalnya_hvac.cooling_signal>0 THEN spalnya_HVAC.fancoil_speed:=1; END_IF

			1:	IF spalnya_hvac.cooling_signal=0 THEN spalnya_HVAC.fancoil_speed:=0; END_IF
				IF spalnya_hvac.cooling_signal>50 THEN  spalnya_HVAC.fancoil_speed:=2; END_IF

			2:	IF spalnya_hvac.cooling_signal=0 THEN spalnya_HVAC.fancoil_speed:=0; END_IF
				IF spalnya_hvac.cooling_signal>75  THEN spalnya_HVAC.fancoil_speed:=3; END_IF
				IF spalnya_hvac.cooling_signal<45  THEN spalnya_HVAC.fancoil_speed:=1; END_IF

			3:	IF spalnya_hvac.cooling_signal=0 THEN spalnya_HVAC.fancoil_speed:=0; END_IF
				IF spalnya_hvac.cooling_signal<75  THEN spalnya_HVAC.fancoil_speed:=2; END_IF
		END_CASE
	END_IF
	IF spalnya_HVAC.cooling_signal = 0 THEN
		CASE spalnya_hvac.fancoil_speed OF
			0:	IF spalnya_hvac.heating_signal>0 THEN spalnya_HVAC.fancoil_speed:=1; END_IF

			1:	IF spalnya_hvac.heating_signal=0 THEN spalnya_HVAC.fancoil_speed:=0; END_IF
				IF spalnya_hvac.heating_signal>50 THEN  spalnya_HVAC.fancoil_speed:=2; END_IF

			2:	IF spalnya_hvac.heating_signal=0 THEN spalnya_HVAC.fancoil_speed:=0; END_IF
				IF spalnya_hvac.heating_signal>75  THEN spalnya_HVAC.fancoil_speed:=3; END_IF
				IF spalnya_hvac.heating_signal<45  THEN spalnya_HVAC.fancoil_speed:=1; END_IF

			3:	IF spalnya_hvac.heating_signal=0 THEN spalnya_HVAC.fancoil_speed:=0; END_IF
				IF spalnya_hvac.heating_signal<75  THEN spalnya_HVAC.fancoil_speed:=2; END_IF
		END_CASE
	END_IF
END_IF
CASE DYTJACHA_HVAC.fancoil_speed OF
	0:	fancoil_dytjacha_low:=FALSE;
		fancoil_dytjacha_med:=FALSE;
		fancoil_dytjacha_high:=FALSE;

	1:	fancoil_dytjacha_low:=TRUE;
		fancoil_dytjacha_med:=FALSE;
		fancoil_dytjacha_high:=FALSE;

	2:	fancoil_dytjacha_low:=FALSE;
		fancoil_dytjacha_med:=TRUE;
		fancoil_dytjacha_high:=FALSE;

	3:	fancoil_dytjacha_low:=FALSE;
		fancoil_dytjacha_med:=FALSE;
		fancoil_dytjacha_high:=TRUE;
END_CASE

CASE SPALNYA_HVAC.fancoil_speed OF
	0:	fancoil_spalnya_low:=FALSE;
		fancoil_spalnya_med:=FALSE;
		fancoil_spalnya_high:=FALSE;

	1:	fancoil_spalnya_low:=TRUE;
		fancoil_spalnya_med:=FALSE;
		fancoil_spalnya_high:=FALSE;

	2:	fancoil_spalnya_low:=FALSE;
		fancoil_spalnya_med:=TRUE;
		fancoil_spalnya_high:=FALSE;

	3:	fancoil_spalnya_low:=FALSE;
		fancoil_spalnya_med:=FALSE;
		fancoil_spalnya_high:=TRUE;
END_CASE
CASE KABINET_HVAC.fancoil_speed OF
	0:	data2floor[0].0:=0; (*запис в масив даних, що відправляються на 2й поверх*)
		data2floor[0].1:=0;
		data2floor[0].2:=0;

	1:	data2floor[0].0:=1; (*запис в масив даних, що відправляються на 2й поверх*)
		data2floor[0].1:=0;
		data2floor[0].2:=0;

	2:	data2floor[0].0:=0; (*запис в масив даних, що відправляються на 2й поверх*)
		data2floor[0].1:=1;
		data2floor[0].2:=0;

	3:	data2floor[0].0:=0; (*запис в масив даних, що відправляються на 2й поверх*)
		data2floor[0].1:=0;
		data2floor[0].2:=1;
END_CASE

CASE KINO_HVAC.fancoil_speed OF
	0:	data2floor[0].3:=0; (*запис в масив даних, що відправляються на 2й поверх*)
		data2floor[0].4:=0;
		data2floor[0].5:=0;

	1:	data2floor[0].3:=1; (*запис в масив даних, що відправляються на 2й поверх*)
		data2floor[0].4:=0;
		data2floor[0].5:=0;

	2:	data2floor[0].3:=0; (*запис в масив даних, що відправляються на 2й поверх*)
		data2floor[0].4:=1;
		data2floor[0].5:=0;

	3:	data2floor[0].3:=0; (*запис в масив даних, що відправляються на 2й поверх*)
		data2floor[0].4:=0;
		data2floor[0].5:=1;
END_CASE

CASE VITALNYA_HVAC.fancoil_speed OF
	0:	data1floor[0].0:=0; (*запис в масив даних, що відправляються на 1й поверх*)
		data1floor[0].1:=0;
		data1floor[0].2:=0;

	1:	data1floor[0].0:=1; (*запис в масив даних, що відправляються на 1й поверх*)
		data1floor[0].1:=0;
		data1floor[0].2:=0;

	2:	data1floor[0].0:=0; (*запис в масив даних, що відправляються на 1й поверх*)
		data1floor[0].1:=1;
		data1floor[0].2:=0;

	3:	data1floor[0].0:=0; (*запис в масив даних, що відправляються на 1й поверх*)
		data1floor[0].1:=0;
		data1floor[0].2:=1;
END_CASE

(*--------------------------------------klapany--------------------------------------------*)
(*data1floor[2]:=WORD_TO_BYTE(VITALNYA_HVAC.klapan); data1floor[3]:=WORD_TO_BYTE(SHR(VITALNYA_HVAC.klapan,8));*)
klapan_vitalnya:=VITALNYA_HVAC.klapan;
klapan_spalnya:=SPALNYA_HVAC.klapan;
klapan_dytjacha:=DYTJACHA_HVAC.klapan;

data2floor[2]:=WORD_TO_BYTE(KABINET_HVAC.klapan); data2floor[3]:=WORD_TO_BYTE(SHR(KABINET_HVAC.klapan,8));
data2floor[4]:=WORD_TO_BYTE(KINO_HVAC.klapan); data2floor[5]:=WORD_TO_BYTE(SHR(KINO_HVAC.klapan,8));

(*------------------------------zaslinky------------------------------------*)
z_vitalnya:=VITALNYA_HVAC.zaslinka;
z_kabinet:=KABINET_HVAC.zaslinka;
z_kino:=KINO_HVAC.zaslinka;
z_dytjacha:=DYTJACHA_HVAC.zaslinka;
z_spalnya:=SPALNYA_HVAC.zaslinka;

(*-----------------------------tepla pidloga-------------------------------*)
data1floor[0].4:=VITALNYA_HVAC.tepla_pidloga;
data2floor[1].0:=KABINET_HVAC.tepla_pidloga;
data2floor[1].1:=KABINET_HVAC.tepla_pidloga;
data2floor[1].2:=STUDIO_HVAC.tepla_pidloga;
data2floor[1].3:=STUDIO_HVAC.tepla_pidloga;

dytjacha_col:=DYTJACHA_HVAC.tepla_pidloga;
spalnya_col:=SPALNYA_HVAC.tepla_pidloga;
END_PROGRAM
ACTION init:
IF i=500 THEN
	t_tamburPrev:=t_tambur_sum/i;
	t_suPrev:=t_su_sum/i;
	t_spalnyaPrev:=t_spalnya_sum/i;
	t_outPrev:=t_out_sum/i;
	t_tambur_sum:=0;
	t_su_sum:=0;
	t_spalnya_sum:=0;
	t_out_sum:=0;
	i:=501;
ELSE
	t_tambur_sum:=t_tambur_sum+temp_tambur*0.1;
	t_su_sum:=t_su_sum+temp_su*0.1;
	t_spalnya_sum:=t_spalnya_sum+temp_spalnya*0.1;
	t_out_sum:=t_out_sum+iT_out*0.1;
	i:=i+1;
END_IF
END_ACTION

(* POU EIB, ST *)
PROGRAM EIB
VAR
	i:INT:=0;
	POWER: EIB_BIT_REC;
	fb_temp_read: EIB_2OCTET_FLOAT_REC;
	fb_read_heating_mode:EIB_BIT_REC;
	fb_req_heating_mode:EIB_READ_SEND;
	fb_setpoint_read:EIB_8BIT_UNSIGN_REC;
	setpoint_vitalnya_dpt4,	setpoint_kino_dpt4,	setpoint_studio_dpt4,	setpoint_kabinet_dpt4,	setpoint_dytjacha_dpt4,	setpoint_spalnya_dpt4:REAL;
	fanspeed_dpt4:REAL;

	fb_heartbeat_timer:TON;
	fb_actual_setpoint_read:EIB_2OCTET_FLOAT_REC;
	fb_actual_setpoint_send:EIB_2OCTET_FLOAT_SEND;
	fb_out_temp_send:EIB_2OCTET_FLOAT_SEND;
	fb_setpoint_switch_send:EIB_BIT_SEND_EX;
	fb_heartbeat_derevo_timer: TON;
	fb_heartbeat1_timer: TON;
	fb_heartbeat2_timer: TON;

	fb_start_delay:TP;

	fb_vitalnya_FCU_cooling_ctrl_sig_rec: EIB_8BIT_UNSIGN_REC;
	fb_kino_FCU_cooling_ctrl_sig_rec: EIB_8BIT_UNSIGN_REC;
	fb_kabinet_FCU_cooling_ctrl_sig_rec: EIB_8BIT_UNSIGN_REC;
	fb_dytjacha_FCU_cooling_ctrl_sig_rec: EIB_8BIT_UNSIGN_REC;
	fb_spalnya_FCU_cooling_ctrl_sig_rec: EIB_8BIT_UNSIGN_REC;

	fb_vitalnya_FCU_heating_ctrl_sig_rec: EIB_8BIT_UNSIGN_REC;
	fb_kino_FCU_heating_ctrl_sig_rec: EIB_8BIT_UNSIGN_REC;
	fb_kabinet_FCU_heating_ctrl_sig_rec: EIB_8BIT_UNSIGN_REC;
	fb_dytjacha_FCU_heating_ctrl_sig_rec: EIB_8BIT_UNSIGN_REC;
	fb_spalnya_FCU_heating_ctrl_sig_rec: EIB_8BIT_UNSIGN_REC;

	fb_vitalnya_FCU_fan_speed_send: EIB_8BIT_UNSIGN_SEND;
	fb_kino_FCU_fan_speed_send: EIB_8BIT_UNSIGN_SEND;
	fb_dytjacha_FCU_fan_speed_send: EIB_8BIT_UNSIGN_SEND;
	fb_spalnya_FCU_fan_speed_send: EIB_8BIT_UNSIGN_SEND;
	fb_kabinet_FCU_fan_speed_send: EIB_8BIT_UNSIGN_SEND;

	fb_vitalnya_damper_ctrl_rec: EIB_BIT_REC;
	fb_kino_damper_ctrl_rec: EIB_BIT_REC;
	fb_kabinet_damper_ctrl_rec: EIB_BIT_REC;
	fb_dytjacha_damper_ctrl_rec: EIB_BIT_REC;
	fb_spalnya_damper_ctrl_rec: EIB_BIT_REC;



	fb_eib_time_rec: EIB_TIME_REC;
	fb_eib_date_rec: EIB_DATE_REC;
	fb_eib_dark_outside_rec: EIB_BIT_REC;
	fb_beckhoff_twillight_send: EIB_BIT_SEND;

	eib_twillight_eib_addr: EIB_GROUP_ADDR := (MAIN:=1,SUB_MAIN:=3,NUMBER:=14);
	b_eib_twillight: BOOL;
	fb_eib_twillight_send: EIB_BIT_SEND;
	fb_eib_twillight_rec: EIB_BIT_REC;
	beckhoff_twillight_eib_addr: EIB_GROUP_ADDR := (MAIN:=1,SUB_MAIN:=3,NUMBER:=13);
END_VAR
fb_start_delay(IN:=  SYSTEMTASKINFOARR[1].firstCycle, PT:=t#60s);
fb_req_heating_mode.bRead:=FALSE;
IF  fb_start_delay.Q THEN
	fb_req_heating_mode(group_address:=heating_mode_addr, str_Rec:=fb_kl6301_0.str_Data_Rec, bread:=fb_start_delay.Q);
END_IF;
fb_read_heating_mode(strData_Rec:=fb_KL6301_0.str_Data_Rec, Group_Address:=heating_mode_addr, bdata=>heating_mode);
(*EIB*)
fb_heartbeat_timer(in:=NOT fb_heartbeat_timer.Q, pt:=t#10s);
fb_KL6301_0.iMode:=1;
CASE i OF
0:	(* EIB Address 2.3.4 *)
	fb_KL6301_0.EIB_PHYS_ADDR.Area:=1;
	fb_KL6301_0.EIB_PHYS_ADDR.Line:=1;
	fb_KL6301_0.EIB_PHYS_ADDR.Device:=1;
	(* Filter 1 *)
	fb_KL6301_0.EIB_GROUP_FILTER[1].GROUP_ADDR.MAIN:=1;
	fb_KL6301_0.EIB_GROUP_FILTER[1].GROUP_ADDR.SUB_MAIN:=1;
	fb_KL6301_0.EIB_GROUP_FILTER[1].GROUP_ADDR.NUMBER:=0;
	fb_KL6301_0.EIB_GROUP_FILTER[1].GROUP_LEN:=31;
	(* Filter 2*)
	fb_KL6301_0.EIB_GROUP_FILTER[2].GROUP_ADDR.MAIN:=1;
	fb_KL6301_0.EIB_GROUP_FILTER[2].GROUP_ADDR.SUB_MAIN:=2;
	fb_KL6301_0.EIB_GROUP_FILTER[2].GROUP_ADDR.NUMBER:=0;
	fb_KL6301_0.EIB_GROUP_FILTER[2].GROUP_LEN:=31;
	(* Filter 3*)
	fb_KL6301_0.EIB_GROUP_FILTER[3].GROUP_ADDR.MAIN:=1;
	fb_KL6301_0.EIB_GROUP_FILTER[3].GROUP_ADDR.SUB_MAIN:=3;
	fb_KL6301_0.EIB_GROUP_FILTER[3].GROUP_ADDR.NUMBER:=0;
	fb_KL6301_0.EIB_GROUP_FILTER[3].GROUP_LEN:=31;
	(* Filter 4 *)
	fb_KL6301_0.EIB_GROUP_FILTER[4].GROUP_ADDR.MAIN:=1;
	fb_KL6301_0.EIB_GROUP_FILTER[4].GROUP_ADDR.SUB_MAIN:=4;
	fb_KL6301_0.EIB_GROUP_FILTER[4].GROUP_ADDR.NUMBER:=0;
	fb_KL6301_0.EIB_GROUP_FILTER[4].GROUP_LEN:=31;
	(* Filter 5*)
	fb_KL6301_0.EIB_GROUP_FILTER[5].GROUP_ADDR.MAIN:=1;
	fb_KL6301_0.EIB_GROUP_FILTER[5].GROUP_ADDR.SUB_MAIN:=5;
	fb_KL6301_0.EIB_GROUP_FILTER[5].GROUP_ADDR.NUMBER:=0;
	fb_KL6301_0.EIB_GROUP_FILTER[5].GROUP_LEN:=31;
	(* Filter 6*)
	fb_KL6301_0.EIB_GROUP_FILTER[6].GROUP_ADDR.MAIN:=1;
	fb_KL6301_0.EIB_GROUP_FILTER[6].GROUP_ADDR.SUB_MAIN:=6;
	fb_KL6301_0.EIB_GROUP_FILTER[6].GROUP_ADDR.NUMBER:=0;
	fb_KL6301_0.EIB_GROUP_FILTER[6].GROUP_LEN:=31;
	(* Filter 7*)
	fb_KL6301_0.EIB_GROUP_FILTER[7].GROUP_ADDR.MAIN:=1;
	fb_KL6301_0.EIB_GROUP_FILTER[7].GROUP_ADDR.SUB_MAIN:=7;
	fb_KL6301_0.EIB_GROUP_FILTER[7].GROUP_ADDR.NUMBER:=0;
	fb_KL6301_0.EIB_GROUP_FILTER[7].GROUP_LEN:=31;
(*	(* Filter 8*)
	fb_KL6301_0.EIB_GROUP_FILTER[8].GROUP_ADDR.MAIN:=1;
	fb_KL6301_0.EIB_GROUP_FILTER[8].GROUP_ADDR.SUB_MAIN:=8;
	fb_KL6301_0.EIB_GROUP_FILTER[8].GROUP_ADDR.NUMBER:=0;
	fb_KL6301_0.EIB_GROUP_FILTER[8].GROUP_LEN:=31;*)

	fb_KL6301_0.bActivate :=TRUE; 	(*Start EIB Functionblock*)
	IF fb_KL6301_0.bReady THEN	(*Wait until the fb is ready *)
		IF NOT fb_KL6301_0.bError THEN
			i:=1;  (* EIB functionblock is now ready to send and receive *)
		ELSE
			i:=100; (* EIB ERROR*)
		END_IF
	END_IF
1:	;
100:	;(*ERROR EIB*)
END_CASE

fb_KL6301_0(
	idx:=1,								(* for every KL6301 an other idx number
										Example KL6301 terminal 1 - idx=1 , KL6301 termnal 2 -idx=3,... max. 64 *)
	KL6301_IN:=KL6301_IN_0,				(* Terminal variable - address IN *)
	KL6301_OUT:=KL6301_OUT_0 );			(* Terminal variable - address OUT *)

fb_out_temp_send(group_address:=out_T_EIB_addr, str_Rec:=fb_kl6301_0.str_Data_Rec, rData:=heat.t_out );



eibPort_climate;

floor3;
floor1;
floor2;
(*derevo_read;*)
derevo;
timers;
END_PROGRAM
ACTION derevo:
fb_derevo_vidpochynok1_read(strData_Rec:=fb_KL6301_0.str_Data_Rec, Group_Address:=derevo_vidpochynok1_adr);
IF NOT  fb_derevo_vidpochynok1_read.bDataReceive THEN
	data_derevo[100].0:= fb_derevo_vidpochynok1_read.bdata;
END_IF

fb_derevo_vidpochynok2_read(strData_Rec:=fb_KL6301_0.str_Data_Rec, Group_Address:=derevo_vidpochynok2_adr);
IF NOT  fb_derevo_vidpochynok2_read.bDataReceive THEN
	data_derevo[100].1:= fb_derevo_vidpochynok2_read.bdata;
END_IF

fb_derevo_veranda_read(strData_Rec:=fb_KL6301_0.str_Data_Rec, Group_Address:=derevo_veranda_adr);
IF NOT  fb_derevo_veranda_read.bDataReceive THEN
	data_derevo[100].2:= fb_derevo_veranda_read.bdata;
END_IF

fb_derevo_veranda_zovn_read(strData_Rec:=fb_KL6301_0.str_Data_Rec, Group_Address:=derevo_veranda_zovn_adr);
IF NOT  fb_derevo_veranda_zovn_read.bDataReceive THEN
	data_derevo[100].3:=fb_derevo_veranda_zovn_read.bdata;
END_IF

fb_derevo_vhid_zovn_read(strData_Rec:=fb_KL6301_0.str_Data_Rec, Group_Address:=derevo_vhid_zovn_adr);
IF NOT  fb_derevo_vhid_zovn_read.bDataReceive THEN
	data_derevo[100].4:= fb_derevo_vhid_zovn_read.bdata;
END_IF

fb_derevo_sauna_read(strData_Rec:=fb_KL6301_0.str_Data_Rec, Group_Address:=derevo_sauna_adr);
IF NOT  fb_derevo_sauna_read.bDataReceive THEN
	data_derevo[100].5:= fb_derevo_sauna_read.bdata;
END_IF

fb_derevo_vhid_read(strData_Rec:=fb_KL6301_0.str_Data_Rec, Group_Address:=derevo_vhid_adr);
IF NOT  fb_derevo_vhid_read.bDataReceive THEN
	data_derevo[100].6:= fb_derevo_vhid_read.bdata;
END_IF

fb_derevo_kotel_read(strData_Rec:=fb_KL6301_0.str_Data_Rec, Group_Address:=derevo_kotel_adr);
IF NOT  fb_derevo_kotel_read.bDataReceive THEN
	data_derevo[100].7:= fb_derevo_kotel_read.bdata;
END_IF

fb_derevo_korydor_read(strData_Rec:=fb_KL6301_0.str_Data_Rec, Group_Address:=derevo_korydor_adr );
IF NOT  fb_derevo_korydor_read.bDataReceive THEN
	data_derevo[101].0:= fb_derevo_korydor_read.bdata;
END_IF
fb_derevo_sinna_read(strData_Rec:=fb_KL6301_0.str_Data_Rec, Group_Address:=derevo_sinna_adr );
IF NOT  fb_derevo_sinna_read.bDataReceive THEN
	data_derevo[101].1:= fb_derevo_sinna_read.bdata;
END_IF
fb_derevo_hamam_read(strData_Rec:=fb_KL6301_0.str_Data_Rec, Group_Address:=derevo_hamam_adr );
IF NOT  fb_derevo_hamam_read.bDataReceive THEN
	data_derevo[101].2:= fb_derevo_hamam_read.bdata;
END_IF
fb_derevo_kuhnya_read(strData_Rec:=fb_KL6301_0.str_Data_Rec, Group_Address:=derevo_kuhnya_adr );
IF NOT  fb_derevo_kuhnya_read.bDataReceive THEN
	data_derevo[101].3:= fb_derevo_kuhnya_read.bdata;
END_IF
fb_derevo_bassein1_read(strData_Rec:=fb_KL6301_0.str_Data_Rec, Group_Address:=derevo_bassein1_adr );
IF NOT  fb_derevo_bassein1_read.bDataReceive THEN
	data_derevo[101].4:= fb_derevo_bassein1_read.bdata;
END_IF
fb_derevo_bassein_lampa_read(strData_Rec:=fb_KL6301_0.str_Data_Rec, Group_Address:=derevo_bassein_lampa_adr );
IF NOT  fb_derevo_bassein_lampa_read.bDataReceive THEN
	data_derevo[101].5:= fb_derevo_bassein_lampa_read.bdata;
END_IF
fb_derevo_spalnya2_read(strData_Rec:=fb_KL6301_0.str_Data_Rec, Group_Address:=derevo_spalnya2_adr);
IF NOT  fb_derevo_spalnya2_read.bDataReceive THEN
	data_derevo[101].6:= fb_derevo_spalnya2_read.bdata;
END_IF
fb_derevo_terassa_read(strData_Rec:=fb_KL6301_0.str_Data_Rec, Group_Address:=derevo_terassa_adr);
IF NOT  fb_derevo_terassa_read.bDataReceive THEN
	data_derevo[101].7:= fb_derevo_terassa_read.bdata;
END_IF
fb_derevo_dush_read(strData_Rec:=fb_KL6301_0.str_Data_Rec, Group_Address:=derevo_dush_adr );
IF NOT  fb_derevo_dush_read.bDataReceive THEN
	data_derevo[102].0:= fb_derevo_dush_read.bdata;
END_IF
fb_derevo_wc_read(strData_Rec:=fb_KL6301_0.str_Data_Rec, Group_Address:=derevo_wc_adr );
IF NOT  fb_derevo_wc_read.bDataReceive THEN
	data_derevo[102].1:= fb_derevo_wc_read.bdata;
END_IF
fb_derevo_spalnya_verh_read(strData_Rec:=fb_KL6301_0.str_Data_Rec, Group_Address:=derevo_spalnya_verh_adr );
IF NOT  fb_derevo_spalnya_verh_read.bDataReceive THEN
	data_derevo[102].2:= fb_derevo_spalnya_verh_read.bdata;
END_IF
fb_derevo_spalnya1_read(strData_Rec:=fb_KL6301_0.str_Data_Rec, Group_Address:=derevo_spalnya1_adr );
IF NOT  fb_derevo_spalnya1_read.bDataReceive THEN
	data_derevo[102].3:= fb_derevo_spalnya1_read.bdata;
END_IF
fb_derevo_spalnya_su_read(strData_Rec:=fb_KL6301_0.str_Data_Rec, Group_Address:=derevo_spalnya_su_adr );
IF NOT  fb_derevo_spalnya_su_read.bDataReceive THEN
	data_derevo[102].4:= fb_derevo_spalnya_su_read.bdata;
END_IF
fb_derevo_garderob_read(strData_Rec:=fb_KL6301_0.str_Data_Rec, Group_Address:=derevo_garderob_adr );
IF NOT  fb_derevo_garderob_read.bDataReceive THEN
	data_derevo[102].5:= fb_derevo_garderob_read.bdata;
END_IF

fb_derevo_dush2_read(strData_Rec:=fb_KL6301_0.str_Data_Rec, Group_Address:=derevo_dush2_adr );
IF NOT  fb_derevo_dush2_read.bDataReceive THEN
	data_derevo[102].6:= fb_derevo_dush2_read.bdata;
END_IF

(*sending*)

fb_derevo_vidpochynok1_send_status_ex(imode:=BOOL_TO_INT(NOT fb_heartbeat_timer.Q)*2, bStart:=fb_heartbeat_timer.IN, str_Rec:=fb_KL6301_0.str_Data_Rec, bData:=derevo_vidpochynok1,  Group_Address:=derevo_vidpochynok1_status_adr);
fb_derevo_vidpochynok2_send_status_ex(imode:=BOOL_TO_INT(NOT fb_heartbeat_timer.Q)*2, bStart:= fb_heartbeat_timer.IN, str_Rec:=fb_KL6301_0.str_Data_Rec, bData:=derevo_vidpochynok2,  Group_Address:=derevo_vidpochynok2_status_adr);
fb_derevo_veranda_send_status_ex(imode:=BOOL_TO_INT(NOT fb_heartbeat_timer.Q)*2, bStart:= fb_heartbeat_timer.IN, str_Rec:=fb_KL6301_0.str_Data_Rec, bData:=derevo_veranda,  Group_Address:=derevo_veranda_status_adr);
fb_derevo_veranda_zovn_send_status_ex(imode:=BOOL_TO_INT(NOT fb_heartbeat_timer.Q)*2, bStart:= fb_heartbeat_timer.IN, str_Rec:=fb_KL6301_0.str_Data_Rec, bData:=derevo_veranda_zovn,  Group_Address:=derevo_veranda_zovn_status_adr);
fb_derevo_sauna_send_status_ex(imode:=BOOL_TO_INT(NOT fb_heartbeat_timer.Q)*2, bStart:= fb_heartbeat_timer.IN, str_Rec:=fb_KL6301_0.str_Data_Rec, bData:=derevo_sauna,  Group_Address:=derevo_sauna_status_adr);
fb_derevo_vhid_zovn_send_status_ex(imode:=BOOL_TO_INT(NOT fb_heartbeat_timer.Q)*2, bStart:= fb_heartbeat_timer.IN, str_Rec:=fb_KL6301_0.str_Data_Rec, bData:=derevo_vhid_zovn,  Group_Address:=derevo_vhid_zovn_status_adr);
fb_derevo_vhid_send_status_ex(imode:=BOOL_TO_INT(NOT fb_heartbeat_timer.Q)*2, bStart:= fb_heartbeat_timer.IN, str_Rec:=fb_KL6301_0.str_Data_Rec, bData:=derevo_vhid,  Group_Address:=derevo_vhid_status_adr);
fb_derevo_kotel_send_status_ex(imode:=BOOL_TO_INT(NOT fb_heartbeat_timer.Q)*2, bStart:= fb_heartbeat_timer.IN, str_Rec:=fb_KL6301_0.str_Data_Rec, bData:=derevo_kotel,  Group_Address:=derevo_kotel_status_adr);
fb_derevo_korydor_send_status_ex(imode:=BOOL_TO_INT(NOT fb_heartbeat_timer.Q)*2, bStart:= fb_heartbeat_timer.IN, str_Rec:=fb_KL6301_0.str_Data_Rec, bData:=derevo_korydor,  Group_Address:=derevo_korydor_status_adr);
fb_derevo_sinna_send_status_ex(imode:=BOOL_TO_INT(NOT fb_heartbeat_timer.Q)*2, bStart:= fb_heartbeat_timer.IN, str_Rec:=fb_KL6301_0.str_Data_Rec, bData:=derevo_sinna,  Group_Address:=derevo_sinna_status_adr);
fb_derevo_hamam_send_status_ex(imode:=BOOL_TO_INT(NOT fb_heartbeat_timer.Q)*2, bStart:= fb_heartbeat_timer.IN, str_Rec:=fb_KL6301_0.str_Data_Rec, bData:=derevo_hamam,  Group_Address:=derevo_hamam_status_adr);
fb_derevo_kuhnya_send_status_ex(imode:=BOOL_TO_INT(NOT fb_heartbeat_timer.Q)*2, bStart:= fb_heartbeat_timer.IN, str_Rec:=fb_KL6301_0.str_Data_Rec, bData:=derevo_kuhnya,  Group_Address:=derevo_kuhnya_status_adr);
fb_derevo_bassein1_send_status_ex(imode:=BOOL_TO_INT(NOT fb_heartbeat_timer.Q)*2, bStart:= fb_heartbeat_timer.IN, str_Rec:=fb_KL6301_0.str_Data_Rec, bData:=derevo_bassein1,  Group_Address:=derevo_bassein1_status_adr);
fb_derevo_bassein_lampa_send_status_ex(imode:=BOOL_TO_INT(NOT fb_heartbeat_timer.Q)*2, bStart:= fb_heartbeat_timer.IN, str_Rec:=fb_KL6301_0.str_Data_Rec, bData:=derevo_bassein_lampa,  Group_Address:=derevo_bassein_lampa_status_adr);
fb_derevo_spalnya2_send_status_ex(imode:=BOOL_TO_INT(NOT fb_heartbeat_timer.Q)*2, bStart:= fb_heartbeat_timer.IN, str_Rec:=fb_KL6301_0.str_Data_Rec, bData:=derevo_spalnya2,  Group_Address:=derevo_spalnya2_status_adr);
fb_derevo_terassa_send_status_ex(imode:=BOOL_TO_INT(NOT fb_heartbeat_timer.Q)*2, bStart:= fb_heartbeat_timer.IN, str_Rec:=fb_KL6301_0.str_Data_Rec, bData:=derevo_terassa,  Group_Address:=derevo_terassa_status_adr);
fb_derevo_dush_send_status_ex(imode:=BOOL_TO_INT(NOT fb_heartbeat_timer.Q)*2, bStart:= fb_heartbeat_timer.IN, str_Rec:=fb_KL6301_0.str_Data_Rec, bData:=derevo_dush,  Group_Address:=derevo_dush_status_adr);
fb_derevo_wc_send_status_ex(imode:=BOOL_TO_INT(NOT fb_heartbeat_timer.Q)*2, bStart:= fb_heartbeat_timer.IN, str_Rec:=fb_KL6301_0.str_Data_Rec, bData:=derevo_wc,  Group_Address:=derevo_wc_status_adr);
fb_derevo_spalnya_verh_send_status_ex(imode:=BOOL_TO_INT(NOT fb_heartbeat_timer.Q)*2, bStart:= fb_heartbeat_timer.IN, str_Rec:=fb_KL6301_0.str_Data_Rec, bData:=derevo_spalnya_verh,  Group_Address:=derevo_spalnya_verh_status_adr);
fb_derevo_spalnya1_send_status_ex(imode:=BOOL_TO_INT(NOT fb_heartbeat_timer.Q)*2, bStart:= fb_heartbeat_timer.IN, str_Rec:=fb_KL6301_0.str_Data_Rec, bData:=derevo_spalnya1,  Group_Address:=derevo_spalnya1_status_adr);
fb_derevo_spalnya_su_send_status_ex(imode:=BOOL_TO_INT(NOT fb_heartbeat_timer.Q)*2, bStart:= fb_heartbeat_timer.IN, str_Rec:=fb_KL6301_0.str_Data_Rec, bData:=derevo_spalnya_su,  Group_Address:=derevo_spalnya_su_status_adr);
fb_derevo_garderob_send_status_ex(imode:=BOOL_TO_INT(NOT fb_heartbeat_timer.Q)*2, bStart:= fb_heartbeat_timer.IN, str_Rec:=fb_KL6301_0.str_Data_Rec, bData:=derevo_garderob,  Group_Address:=derevo_garderob_status_adr);
fb_derevo_dush2_send_status_ex(imode:=BOOL_TO_INT(NOT fb_heartbeat_timer.Q)*2, bStart:= fb_heartbeat_timer.IN, str_Rec:=fb_KL6301_0.str_Data_Rec, bData:=derevo_dush2,  Group_Address:=derevo_dush2_status_adr);

IF fb_derevo_vidpochynok1_send_status_ex.bSend  THEN
	data_derevo[100].0:=derevo_vidpochynok1;
END_IF

IF fb_derevo_vidpochynok2_send_status_ex.bSend THEN
	data_derevo[100].1:=derevo_vidpochynok2;
END_IF

IF fb_derevo_veranda_send_status_ex.bSend THEN
	data_derevo[100].2:=derevo_veranda;
END_IF

IF fb_derevo_veranda_send_status_ex.bSend THEN
	data_derevo[100].2:=derevo_veranda;
END_IF

IF fb_derevo_veranda_zovn_send_status_ex.bSend   THEN
	data_derevo[100].3:=derevo_veranda_zovn;
END_IF

IF fb_derevo_vhid_zovn_send_status_ex.bSend THEN
	data_derevo[100].4:=derevo_vhid_zovn;
END_IF

IF fb_derevo_sauna_send_status_ex.bSend THEN
	data_derevo[100].5:=derevo_sauna;
END_IF

IF fb_derevo_vhid_send_status_ex.bSend THEN
	data_derevo[100].6:=derevo_vhid;
END_IF

IF fb_derevo_kotel_send_status_ex.bSend THEN
	data_derevo[100].7:=derevo_kotel;
END_IF

IF fb_derevo_korydor_send_status_ex.bSend THEN
	data_derevo[101].0:=derevo_korydor;
END_IF

IF fb_derevo_sinna_send_status_ex.bSend THEN
	data_derevo[101].1:=derevo_sinna;
END_IF

IF fb_derevo_hamam_send_status_ex.bSend THEN
	data_derevo[101].2:=derevo_hamam;
END_IF

IF fb_derevo_kuhnya_send_status_ex.bSend THEN
	data_derevo[101].3:=derevo_kuhnya;
END_IF

IF fb_derevo_bassein1_send_status_ex.bSend THEN
	data_derevo[101].4:=derevo_bassein1;
END_IF

IF fb_derevo_bassein_lampa_send_status_ex.bSend THEN
	data_derevo[101].5:=derevo_bassein_lampa;
END_IF

IF fb_derevo_spalnya2_send_status_ex.bSend THEN
	data_derevo[101].6:=derevo_spalnya2;
END_IF

IF fb_derevo_terassa_send_status_ex.bSend THEN
	data_derevo[101].7:=derevo_terassa;
END_IF

IF fb_derevo_dush_send_status_ex.bSend THEN
	data_derevo[102].0:=derevo_dush;
END_IF

IF fb_derevo_wc_send_status_ex.bSend THEN
	data_derevo[102].1:=derevo_wc;
END_IF

IF fb_derevo_spalnya_verh_send_status_ex.bSend THEN
	data_derevo[102].2:=derevo_spalnya_verh;
END_IF

IF fb_derevo_spalnya1_send_status_ex.bSend THEN
	data_derevo[102].3:=derevo_spalnya1;
END_IF

IF fb_derevo_spalnya_su_send_status_ex.bSend THEN
	data_derevo[102].4:=derevo_spalnya_su;
END_IF

IF fb_derevo_garderob_send_status_ex.bSend THEN
	data_derevo[102].5:=derevo_garderob;
END_IF

